    (* Table initialization: fTable_Be *)
    fTable_Be[0, 0] := 10.0000; fTable_Be[0, 1] := -9999; fTable_Be[0, 2] := 1.70333;
    fTable_Be[1, 0] := 10.1617; fTable_Be[1, 1] := -9999; fTable_Be[1, 2] := 1.71802;
    fTable_Be[2, 0] := 10.3261; fTable_Be[2, 1] := -9999; fTable_Be[2, 2] := 1.73284;
    fTable_Be[3, 0] := 10.4931; fTable_Be[3, 1] := -9999; fTable_Be[3, 2] := 1.74778;
    fTable_Be[4, 0] := 10.6628; fTable_Be[4, 1] := -9999; fTable_Be[4, 2] := 1.75737;
    fTable_Be[5, 0] := 10.8353; fTable_Be[5, 1] := -9999; fTable_Be[5, 2] := 1.76678;
    fTable_Be[6, 0] := 11.0105; fTable_Be[6, 1] := -9999; fTable_Be[6, 2] := 1.77624;
    fTable_Be[7, 0] := 11.1886; fTable_Be[7, 1] := -9999; fTable_Be[7, 2] := 1.78574;
    fTable_Be[8, 0] := 11.3696; fTable_Be[8, 1] := -9999; fTable_Be[8, 2] := 1.79530;
    fTable_Be[9, 0] := 11.5535; fTable_Be[9, 1] := -9999; fTable_Be[9, 2] := 1.80306;
    fTable_Be[10, 0] := 11.7404; fTable_Be[10, 1] := -9999; fTable_Be[10, 2] := 1.80629;
    fTable_Be[11, 0] := 11.9303; fTable_Be[11, 1] := -9999; fTable_Be[11, 2] := 1.80952;
    fTable_Be[12, 0] := 12.1232; fTable_Be[12, 1] := -9999; fTable_Be[12, 2] := 1.81276;
    fTable_Be[13, 0] := 12.3193; fTable_Be[13, 1] := -9999; fTable_Be[13, 2] := 1.81600;
    fTable_Be[14, 0] := 12.5186; fTable_Be[14, 1] := -9999; fTable_Be[14, 2] := 1.81871;
    fTable_Be[15, 0] := 12.7210; fTable_Be[15, 1] := -9999; fTable_Be[15, 2] := 1.81609;
    fTable_Be[16, 0] := 12.9268; fTable_Be[16, 1] := -9999; fTable_Be[16, 2] := 1.81347;
    fTable_Be[17, 0] := 13.1359; fTable_Be[17, 1] := -9999; fTable_Be[17, 2] := 1.80922;
    fTable_Be[18, 0] := 13.3483; fTable_Be[18, 1] := -9999; fTable_Be[18, 2] := 1.80410;
    fTable_Be[19, 0] := 13.5642; fTable_Be[19, 1] := -9999; fTable_Be[19, 2] := 1.79747;
    fTable_Be[20, 0] := 13.7836; fTable_Be[20, 1] := -9999; fTable_Be[20, 2] := 1.78729;
    fTable_Be[21, 0] := 14.0066; fTable_Be[21, 1] := -9999; fTable_Be[21, 2] := 1.77705;
    fTable_Be[22, 0] := 14.2331; fTable_Be[22, 1] := -9999; fTable_Be[22, 2] := 1.76267;
    fTable_Be[23, 0] := 14.4633; fTable_Be[23, 1] := -9999; fTable_Be[23, 2] := 1.74841;
    fTable_Be[24, 0] := 14.6972; fTable_Be[24, 1] := -9999; fTable_Be[24, 2] := 1.72956;
    fTable_Be[25, 0] := 14.9350; fTable_Be[25, 1] := -9999; fTable_Be[25, 2] := 1.71004;
    fTable_Be[26, 0] := 15.1765; fTable_Be[26, 1] := -9999; fTable_Be[26, 2] := 1.68541;
    fTable_Be[27, 0] := 15.4220; fTable_Be[27, 1] := -9999; fTable_Be[27, 2] := 1.65917;
    fTable_Be[28, 0] := 15.6714; fTable_Be[28, 1] := -9999; fTable_Be[28, 2] := 1.62778;
    fTable_Be[29, 0] := 15.9249; fTable_Be[29, 1] := -9999; fTable_Be[29, 2] := 1.59448;
    fTable_Be[30, 0] := 16.1825; fTable_Be[30, 1] := -9999; fTable_Be[30, 2] := 1.55788;
    fTable_Be[31, 0] := 16.4442; fTable_Be[31, 1] := -9999; fTable_Be[31, 2] := 1.52050;
    fTable_Be[32, 0] := 16.7102; fTable_Be[32, 1] := -9999; fTable_Be[32, 2] := 1.47675;
    fTable_Be[33, 0] := 16.9805; fTable_Be[33, 1] := -9999; fTable_Be[33, 2] := 1.43237;
    fTable_Be[34, 0] := 17.2551; fTable_Be[34, 1] := -9999; fTable_Be[34, 2] := 1.38176;
    fTable_Be[35, 0] := 17.5342; fTable_Be[35, 1] := -9999; fTable_Be[35, 2] := 1.33102;
    fTable_Be[36, 0] := 17.8178; fTable_Be[36, 1] := -9999; fTable_Be[36, 2] := 1.27265;
    fTable_Be[37, 0] := 18.1060; fTable_Be[37, 1] := -9999; fTable_Be[37, 2] := 1.22588;
    fTable_Be[38, 0] := 18.3988; fTable_Be[38, 1] := -9999; fTable_Be[38, 2] := 1.19605;
    fTable_Be[39, 0] := 18.6964; fTable_Be[39, 1] := -9999; fTable_Be[39, 2] := 1.16961;
    fTable_Be[40, 0] := 18.9988; fTable_Be[40, 1] := -9999; fTable_Be[40, 2] := 1.14509;
    fTable_Be[41, 0] := 19.3061; fTable_Be[41, 1] := 2.30967; fTable_Be[41, 2] := 1.10518;
    fTable_Be[42, 0] := 19.6184; fTable_Be[42, 1] := 2.31367; fTable_Be[42, 2] := 1.06950;
    fTable_Be[43, 0] := 19.9357; fTable_Be[43, 1] := 2.31537; fTable_Be[43, 2] := 1.03964;
    fTable_Be[44, 0] := 20.2581; fTable_Be[44, 1] := 2.31755; fTable_Be[44, 2] := 1.01722;
    fTable_Be[45, 0] := 20.5858; fTable_Be[45, 1] := 2.32374; fTable_Be[45, 2] := 0.999039;
    fTable_Be[46, 0] := 20.9187; fTable_Be[46, 1] := 2.34045; fTable_Be[46, 2] := 0.987135;
    fTable_Be[47, 0] := 21.2571; fTable_Be[47, 1] := 2.37239; fTable_Be[47, 2] := 0.952742;
    fTable_Be[48, 0] := 21.6009; fTable_Be[48, 1] := 2.38699; fTable_Be[48, 2] := 0.912693;
    fTable_Be[49, 0] := 21.9503; fTable_Be[49, 1] := 2.39600; fTable_Be[49, 2] := 0.874329;
    fTable_Be[50, 0] := 22.3053; fTable_Be[50, 1] := 2.40177; fTable_Be[50, 2] := 0.837576;
    fTable_Be[51, 0] := 22.6661; fTable_Be[51, 1] := 2.40538; fTable_Be[51, 2] := 0.802368;
    fTable_Be[52, 0] := 23.0327; fTable_Be[52, 1] := 2.40746; fTable_Be[52, 2] := 0.768641;
    fTable_Be[53, 0] := 23.4052; fTable_Be[53, 1] := 2.40846; fTable_Be[53, 2] := 0.736331;
    fTable_Be[54, 0] := 23.7838; fTable_Be[54, 1] := 2.40939; fTable_Be[54, 2] := 0.705380;
    fTable_Be[55, 0] := 24.1685; fTable_Be[55, 1] := 2.41248; fTable_Be[55, 2] := 0.675729;
    fTable_Be[56, 0] := 24.5594; fTable_Be[56, 1] := 2.41570; fTable_Be[56, 2] := 0.647325;
    fTable_Be[57, 0] := 24.9566; fTable_Be[57, 1] := 2.42027; fTable_Be[57, 2] := 0.609275;
    fTable_Be[58, 0] := 25.3602; fTable_Be[58, 1] := 2.41808; fTable_Be[58, 2] := 0.567900;
    fTable_Be[59, 0] := 25.7704; fTable_Be[59, 1] := 2.40985; fTable_Be[59, 2] := 0.529334;
    fTable_Be[60, 0] := 26.1872; fTable_Be[60, 1] := 2.39826; fTable_Be[60, 2] := 0.493388;
    fTable_Be[61, 0] := 26.6108; fTable_Be[61, 1] := 2.38435; fTable_Be[61, 2] := 0.459883;
    fTable_Be[62, 0] := 27.0412; fTable_Be[62, 1] := 2.36859; fTable_Be[62, 2] := 0.428653;
    fTable_Be[63, 0] := 27.4786; fTable_Be[63, 1] := 2.35116; fTable_Be[63, 2] := 0.399544;
    fTable_Be[64, 0] := 27.9230; fTable_Be[64, 1] := 2.33226; fTable_Be[64, 2] := 0.372411;
    fTable_Be[65, 0] := 28.3747; fTable_Be[65, 1] := 2.30996; fTable_Be[65, 2] := 0.347121;
    fTable_Be[66, 0] := 28.8336; fTable_Be[66, 1] := 2.28594; fTable_Be[66, 2] := 0.328404;
    fTable_Be[67, 0] := 29.3000; fTable_Be[67, 1] := 2.26312; fTable_Be[67, 2] := 0.315229;
    fTable_Be[68, 0] := 29.7739; fTable_Be[68, 1] := 2.24541; fTable_Be[68, 2] := 0.302582;
    fTable_Be[69, 0] := 30.2554; fTable_Be[69, 1] := 2.22901; fTable_Be[69, 2] := 0.290443;
    fTable_Be[70, 0] := 30.7448; fTable_Be[70, 1] := 2.21325; fTable_Be[70, 2] := 0.278791;
    fTable_Be[71, 0] := 31.2421; fTable_Be[71, 1] := 2.19800; fTable_Be[71, 2] := 0.267606;
    fTable_Be[72, 0] := 31.7474; fTable_Be[72, 1] := 2.18311; fTable_Be[72, 2] := 0.256870;
    fTable_Be[73, 0] := 32.2609; fTable_Be[73, 1] := 2.16844; fTable_Be[73, 2] := 0.246565;
    fTable_Be[74, 0] := 32.7827; fTable_Be[74, 1] := 2.15391; fTable_Be[74, 2] := 0.236673;
    fTable_Be[75, 0] := 33.3129; fTable_Be[75, 1] := 2.13952; fTable_Be[75, 2] := 0.227178;
    fTable_Be[76, 0] := 33.8517; fTable_Be[76, 1] := 2.12325; fTable_Be[76, 2] := 0.218064;
    fTable_Be[77, 0] := 34.3992; fTable_Be[77, 1] := 2.10677; fTable_Be[77, 2] := 0.211374;
    fTable_Be[78, 0] := 34.9556; fTable_Be[78, 1] := 2.09142; fTable_Be[78, 2] := 0.206573;
    fTable_Be[79, 0] := 35.5210; fTable_Be[79, 1] := 2.07852; fTable_Be[79, 2] := 0.201882;
    fTable_Be[80, 0] := 36.0955; fTable_Be[80, 1] := 2.06586; fTable_Be[80, 2] := 0.197297;
    fTable_Be[81, 0] := 36.6793; fTable_Be[81, 1] := 2.05353; fTable_Be[81, 2] := 0.192816;
    fTable_Be[82, 0] := 37.2726; fTable_Be[82, 1] := 2.04141; fTable_Be[82, 2] := 0.188437;
    fTable_Be[83, 0] := 37.8754; fTable_Be[83, 1] := 2.02931; fTable_Be[83, 2] := 0.184157;
    fTable_Be[84, 0] := 38.4880; fTable_Be[84, 1] := 2.01697; fTable_Be[84, 2] := 0.179975;
    fTable_Be[85, 0] := 38.9000; fTable_Be[85, 1] := 2.00799; fTable_Be[85, 2] := 0.177252;
    fTable_Be[86, 0] := 39.2000; fTable_Be[86, 1] := 2.00121; fTable_Be[86, 2] := 0.176713;
    fTable_Be[87, 0] := 39.5000; fTable_Be[87, 1] := 1.99567; fTable_Be[87, 2] := 0.176983;
    fTable_Be[88, 0] := 39.9000; fTable_Be[88, 1] := 1.98913; fTable_Be[88, 2] := 0.175827;
    fTable_Be[89, 0] := 40.0000; fTable_Be[89, 1] := 1.98733; fTable_Be[89, 2] := 0.175565;
    fTable_Be[90, 0] := 40.2760; fTable_Be[90, 1] := 1.98264; fTable_Be[90, 2] := 0.174663;
    fTable_Be[91, 0] := 40.5560; fTable_Be[91, 1] := 1.97786; fTable_Be[91, 2] := 0.174609;
    fTable_Be[92, 0] := 40.6970; fTable_Be[92, 1] := 1.97610; fTable_Be[92, 2] := 0.174013;
    fTable_Be[93, 0] := 41.1270; fTable_Be[93, 1] := 1.96960; fTable_Be[93, 2] := 0.173456;
    fTable_Be[94, 0] := 41.5660; fTable_Be[94, 1] := 1.96327; fTable_Be[94, 2] := 0.171435;
    fTable_Be[95, 0] := 42.1670; fTable_Be[95, 1] := 1.95400; fTable_Be[95, 2] := 0.170039;
    fTable_Be[96, 0] := 42.4730; fTable_Be[96, 1] := 1.94966; fTable_Be[96, 2] := 0.168799;
    fTable_Be[97, 0] := 42.9420; fTable_Be[97, 1] := 1.94280; fTable_Be[97, 2] := 0.168198;
    fTable_Be[98, 0] := 43.2600; fTable_Be[98, 1] := 1.93854; fTable_Be[98, 2] := 0.166905;
    fTable_Be[99, 0] := 43.7460; fTable_Be[99, 1] := 1.93138; fTable_Be[99, 2] := 0.165791;
    fTable_Be[100, 0] := 44.0760; fTable_Be[100, 1] := 1.92708; fTable_Be[100, 2] := 0.165390;
    fTable_Be[101, 0] := 44.4110; fTable_Be[101, 1] := 1.92291; fTable_Be[101, 2] := 0.164383;
    fTable_Be[102, 0] := 44.5810; fTable_Be[102, 1] := 1.92070; fTable_Be[102, 2] := 0.163618;
    fTable_Be[103, 0] := 44.9240; fTable_Be[103, 1] := 1.91607; fTable_Be[103, 2] := 0.162962;
    fTable_Be[104, 0] := 45.2720; fTable_Be[104, 1] := 1.91126; fTable_Be[104, 2] := 0.161326;
    fTable_Be[105, 0] := 45.4480; fTable_Be[105, 1] := 1.90903; fTable_Be[105, 2] := 0.161038;
    fTable_Be[106, 0] := 45.9850; fTable_Be[106, 1] := 1.90129; fTable_Be[106, 2] := 0.159149;
    fTable_Be[107, 0] := 46.7288; fTable_Be[107, 1] := 1.89036; fTable_Be[107, 2] := 0.157516;
    fTable_Be[108, 0] := 47.4846; fTable_Be[108, 1] := 1.87948; fTable_Be[108, 2] := 0.155990;
    fTable_Be[109, 0] := 47.6740; fTable_Be[109, 1] := 1.87667; fTable_Be[109, 2] := 0.155621;
    fTable_Be[110, 0] := 48.2650; fTable_Be[110, 1] := 1.86782; fTable_Be[110, 2] := 0.155028;
    fTable_Be[111, 0] := 48.8710; fTable_Be[111, 1] := 1.85943; fTable_Be[111, 2] := 0.155666;
    fTable_Be[112, 0] := 49.0760; fTable_Be[112, 1] := 1.85755; fTable_Be[112, 2] := 0.155951;
    fTable_Be[113, 0] := 49.2830; fTable_Be[113, 1] := 1.85503; fTable_Be[113, 2] := 0.154508;
    fTable_Be[114, 0] := 49.8930; fTable_Be[114, 1] := 1.84657; fTable_Be[114, 2] := 0.154198;
    fTable_Be[115, 0] := 50.7000; fTable_Be[115, 1] := 1.83364; fTable_Be[115, 2] := 0.155814;
    fTable_Be[116, 0] := 51.5200; fTable_Be[116, 1] := 1.82367; fTable_Be[116, 2] := 0.157447;
    fTable_Be[117, 0] := 51.9010; fTable_Be[117, 1] := 1.81956; fTable_Be[117, 2] := 0.158203;
    fTable_Be[118, 0] := 52.4010; fTable_Be[118, 1] := 1.81434; fTable_Be[118, 2] := 0.158683;
    fTable_Be[119, 0] := 53.2485; fTable_Be[119, 1] := 1.80585; fTable_Be[119, 2] := 0.158768;
    fTable_Be[120, 0] := 53.4010; fTable_Be[120, 1] := 1.80449; fTable_Be[120, 2] := 0.158784;
    fTable_Be[121, 0] := 53.9000; fTable_Be[121, 1] := 1.79914; fTable_Be[121, 2] := 0.157647;
    fTable_Be[122, 0] := 54.4010; fTable_Be[122, 1] := 1.79325; fTable_Be[122, 2] := 0.156933;
    fTable_Be[123, 0] := 54.9010; fTable_Be[123, 1] := 1.78748; fTable_Be[123, 2] := 0.157035;
    fTable_Be[124, 0] := 55.4000; fTable_Be[124, 1] := 1.78219; fTable_Be[124, 2] := 0.156125;
    fTable_Be[125, 0] := 55.9010; fTable_Be[125, 1] := 1.77644; fTable_Be[125, 2] := 0.155633;
    fTable_Be[126, 0] := 56.8052; fTable_Be[126, 1] := 1.76616; fTable_Be[126, 2] := 0.152967;
    fTable_Be[127, 0] := 56.9010; fTable_Be[127, 1] := 1.76491; fTable_Be[127, 2] := 0.152689;
    fTable_Be[128, 0] := 57.4010; fTable_Be[128, 1] := 1.75779; fTable_Be[128, 2] := 0.151560;
    fTable_Be[129, 0] := 57.9010; fTable_Be[129, 1] := 1.75138; fTable_Be[129, 2] := 0.151256;
    fTable_Be[130, 0] := 58.4000; fTable_Be[130, 1] := 1.74467; fTable_Be[130, 2] := 0.149795;
    fTable_Be[131, 0] := 59.3446; fTable_Be[131, 1] := 1.73066; fTable_Be[131, 2] := 0.148143;
    fTable_Be[132, 0] := 60.3044; fTable_Be[132, 1] := 1.71666; fTable_Be[132, 2] := 0.147555;
    fTable_Be[133, 0] := 60.9010; fTable_Be[133, 1] := 1.70803; fTable_Be[133, 2] := 0.147236;
    fTable_Be[134, 0] := 61.4010; fTable_Be[134, 1] := 1.70036; fTable_Be[134, 2] := 0.146656;
    fTable_Be[135, 0] := 62.3941; fTable_Be[135, 1] := 1.68542; fTable_Be[135, 2] := 0.147197;
    fTable_Be[136, 0] := 62.4010; fTable_Be[136, 1] := 1.68532; fTable_Be[136, 2] := 0.147201;
    fTable_Be[137, 0] := 63.4000; fTable_Be[137, 1] := 1.67044; fTable_Be[137, 2] := 0.146706;
    fTable_Be[138, 0] := 63.9020; fTable_Be[138, 1] := 1.66247; fTable_Be[138, 2] := 0.147388;
    fTable_Be[139, 0] := 64.4000; fTable_Be[139, 1] := 1.65492; fTable_Be[139, 2] := 0.147185;
    fTable_Be[140, 0] := 65.4010; fTable_Be[140, 1] := 1.63983; fTable_Be[140, 2] := 0.147806;
    fTable_Be[141, 0] := 65.9010; fTable_Be[141, 1] := 1.63182; fTable_Be[141, 2] := 0.147426;
    fTable_Be[142, 0] := 66.9669; fTable_Be[142, 1] := 1.61497; fTable_Be[142, 2] := 0.147801;
    fTable_Be[143, 0] := 68.0500; fTable_Be[143, 1] := 1.59766; fTable_Be[143, 2] := 0.147747;
    fTable_Be[144, 0] := 69.1507; fTable_Be[144, 1] := 1.57948; fTable_Be[144, 2] := 0.147404;
    fTable_Be[145, 0] := 69.4010; fTable_Be[145, 1] := 1.57524; fTable_Be[145, 2] := 0.147327;
    fTable_Be[146, 0] := 70.2340; fTable_Be[146, 1] := 1.56001; fTable_Be[146, 2] := 0.145950;
    fTable_Be[147, 0] := 71.3700; fTable_Be[147, 1] := 1.53888; fTable_Be[147, 2] := 0.145981;
    fTable_Be[148, 0] := 72.5243; fTable_Be[148, 1] := 1.51676; fTable_Be[148, 2] := 0.146011;
    fTable_Be[149, 0] := 72.5670; fTable_Be[149, 1] := 1.51586; fTable_Be[149, 2] := 0.146012;
    fTable_Be[150, 0] := 72.9000; fTable_Be[150, 1] := 1.50929; fTable_Be[150, 2] := 0.145632;
    fTable_Be[151, 0] := 73.5680; fTable_Be[151, 1] := 1.49567; fTable_Be[151, 2] := 0.146079;
    fTable_Be[152, 0] := 74.7579; fTable_Be[152, 1] := 1.47049; fTable_Be[152, 2] := 0.146106;
    fTable_Be[153, 0] := 74.9000; fTable_Be[153, 1] := 1.46741; fTable_Be[153, 2] := 0.146109;
    fTable_Be[154, 0] := 75.2350; fTable_Be[154, 1] := 1.46015; fTable_Be[154, 2] := 0.146426;
    fTable_Be[155, 0] := 75.5670; fTable_Be[155, 1] := 1.45305; fTable_Be[155, 2] := 0.146447;
    fTable_Be[156, 0] := 76.5680; fTable_Be[156, 1] := 1.43052; fTable_Be[156, 2] := 0.147310;
    fTable_Be[157, 0] := 77.2350; fTable_Be[157, 1] := 1.41539; fTable_Be[157, 2] := 0.147639;
    fTable_Be[158, 0] := 77.5670; fTable_Be[158, 1] := 1.40764; fTable_Be[158, 2] := 0.148124;
    fTable_Be[159, 0] := 77.9010; fTable_Be[159, 1] := 1.40006; fTable_Be[159, 2] := 0.148179;
    fTable_Be[160, 0] := 78.5670; fTable_Be[160, 1] := 1.38396; fTable_Be[160, 2] := 0.148938;
    fTable_Be[161, 0] := 78.9000; fTable_Be[161, 1] := 1.37631; fTable_Be[161, 2] := 0.148969;
    fTable_Be[162, 0] := 80.1761; fTable_Be[162, 1] := 1.34408; fTable_Be[162, 2] := 0.150222;
    fTable_Be[163, 0] := 80.9000; fTable_Be[163, 1] := 1.32524; fTable_Be[163, 2] := 0.150928;
    fTable_Be[164, 0] := 81.2340; fTable_Be[164, 1] := 1.31669; fTable_Be[164, 2] := 0.151099;
    fTable_Be[165, 0] := 81.5680; fTable_Be[165, 1] := 1.30817; fTable_Be[165, 2] := 0.151573;
    fTable_Be[166, 0] := 82.8873; fTable_Be[166, 1] := 1.27205; fTable_Be[166, 2] := 0.152380;
    fTable_Be[167, 0] := 83.5680; fTable_Be[167, 1] := 1.25273; fTable_Be[167, 2] := 0.152793;
    fTable_Be[168, 0] := 84.9010; fTable_Be[168, 1] := 1.21283; fTable_Be[168, 2] := 0.152919;
    fTable_Be[169, 0] := 86.2742; fTable_Be[169, 1] := 1.16875; fTable_Be[169, 2] := 0.153088;
    fTable_Be[170, 0] := 87.6696; fTable_Be[170, 1] := 1.12068; fTable_Be[170, 2] := 0.152944;
    fTable_Be[171, 0] := 89.0876; fTable_Be[171, 1] := 1.06780; fTable_Be[171, 2] := 0.152717;
    fTable_Be[172, 0] := 90.5285; fTable_Be[172, 1] := 1.00938; fTable_Be[172, 2] := 0.152457;
    fTable_Be[173, 0] := 91.9928; fTable_Be[173, 1] := 0.944630; fTable_Be[173, 2] := 0.152189;
    fTable_Be[174, 0] := 93.4807; fTable_Be[174, 1] := 0.872376; fTable_Be[174, 2] := 0.151920;
    fTable_Be[175, 0] := 94.9926; fTable_Be[175, 1] := 0.791324; fTable_Be[175, 2] := 0.151867;
    fTable_Be[176, 0] := 96.5291; fTable_Be[176, 1] := 0.699761; fTable_Be[176, 2] := 0.151828;
    fTable_Be[177, 0] := 97.5670; fTable_Be[177, 1] := 0.631310; fTable_Be[177, 2] := 0.151801;
    fTable_Be[178, 0] := 98.5680; fTable_Be[178, 1] := 0.560328; fTable_Be[178, 2] := 0.152508;
    fTable_Be[179, 0] := 98.7770; fTable_Be[179, 1] := 0.544993; fTable_Be[179, 2] := 0.152245;
    fTable_Be[180, 0] := 99.5260; fTable_Be[180, 1] := 0.486543; fTable_Be[180, 2] := 0.151861;
    fTable_Be[181, 0] := 99.9010; fTable_Be[181, 1] := 0.455599; fTable_Be[181, 2] := 0.151904;
    fTable_Be[182, 0] := 100.270; fTable_Be[182, 1] := 0.424344; fTable_Be[182, 2] := 0.151744;
    fTable_Be[183, 0] := 100.660; fTable_Be[183, 1] := 0.389731; fTable_Be[183, 2] := 0.152054;
    fTable_Be[184, 0] := 102.030; fTable_Be[184, 1] := 0.258588; fTable_Be[184, 2] := 0.151656;
    fTable_Be[185, 0] := 102.400; fTable_Be[185, 1] := 0.219148; fTable_Be[185, 2] := 0.151818;
    fTable_Be[186, 0] := 103.770; fTable_Be[186, 1] := 0.0597848; fTable_Be[186, 2] := 0.151969;
    fTable_Be[187, 0] := 104.030; fTable_Be[187, 1] := 0.0260858; fTable_Be[187, 2] := 0.152169;
    fTable_Be[188, 0] := 105.530; fTable_Be[188, 1] := -0.191568; fTable_Be[188, 2] := 0.151371;
    fTable_Be[189, 0] := 106.530; fTable_Be[189, 1] := -0.368308; fTable_Be[189, 2] := 0.151676;
    fTable_Be[190, 0] := 106.900; fTable_Be[190, 1] := -0.441904; fTable_Be[190, 2] := 0.152246;
    fTable_Be[191, 0] := 107.770; fTable_Be[191, 1] := -0.637412; fTable_Be[191, 2] := 0.154099;
    fTable_Be[192, 0] := 108.030; fTable_Be[192, 1] := -0.702374; fTable_Be[192, 2] := 0.155662;
    fTable_Be[193, 0] := 108.280; fTable_Be[193, 1] := -0.768299; fTable_Be[193, 2] := 0.156220;
    fTable_Be[194, 0] := 108.400; fTable_Be[194, 1] := -0.802126; fTable_Be[194, 2] := 0.155741;
    fTable_Be[195, 0] := 108.530; fTable_Be[195, 1] := -0.840651; fTable_Be[195, 2] := 0.156004;
    fTable_Be[196, 0] := 108.650; fTable_Be[196, 1] := -0.876311; fTable_Be[196, 2] := 0.158215;
    fTable_Be[197, 0] := 108.770; fTable_Be[197, 1] := -0.912731; fTable_Be[197, 2] := 0.158122;
    fTable_Be[198, 0] := 109.030; fTable_Be[198, 1] := -0.997553; fTable_Be[198, 2] := 0.159793;
    fTable_Be[199, 0] := 109.150; fTable_Be[199, 1] := -1.03849; fTable_Be[199, 2] := 0.161052;
    fTable_Be[200, 0] := 109.270; fTable_Be[200, 1] := -1.08113; fTable_Be[200, 2] := 0.161306;
    fTable_Be[201, 0] := 109.400; fTable_Be[201, 1] := -1.12894; fTable_Be[201, 2] := 0.163454;
    fTable_Be[202, 0] := 109.530; fTable_Be[202, 1] := -1.17915; fTable_Be[202, 2] := 0.163557;
    fTable_Be[203, 0] := 109.770; fTable_Be[203, 1] := -1.27829; fTable_Be[203, 2] := 0.165902;
    fTable_Be[204, 0] := 109.900; fTable_Be[204, 1] := -1.33524; fTable_Be[204, 2] := 0.168057;
    fTable_Be[205, 0] := 110.030; fTable_Be[205, 1] := -1.39580; fTable_Be[205, 2] := 0.168777;
    fTable_Be[206, 0] := 110.160; fTable_Be[206, 1] := -1.45968; fTable_Be[206, 2] := 0.171253;
    fTable_Be[207, 0] := 110.270; fTable_Be[207, 1] := -1.51640; fTable_Be[207, 2] := 0.172992;
    fTable_Be[208, 0] := 110.530; fTable_Be[208, 1] := -1.66366; fTable_Be[208, 2] := 0.176080;
    fTable_Be[209, 0] := 110.660; fTable_Be[209, 1] := -1.74613; fTable_Be[209, 2] := 0.179584;
    fTable_Be[210, 0] := 110.770; fTable_Be[210, 1] := -1.81926; fTable_Be[210, 2] := 0.183052;
    fTable_Be[211, 0] := 110.900; fTable_Be[211, 1] := -1.91441; fTable_Be[211, 2] := 0.183759;
    fTable_Be[212, 0] := 111.030; fTable_Be[212, 1] := -2.01892; fTable_Be[212, 2] := 0.188659;
    fTable_Be[213, 0] := 111.150; fTable_Be[213, 1] := -2.12502; fTable_Be[213, 2] := 0.191441;
    fTable_Be[214, 0] := 111.280; fTable_Be[214, 1] := -2.25725; fTable_Be[214, 2] := 0.192239;
    fTable_Be[215, 0] := 111.400; fTable_Be[215, 1] := -2.40087; fTable_Be[215, 2] := 0.199075;
    fTable_Be[216, 0] := 111.530; fTable_Be[216, 1] := -2.58708; fTable_Be[216, 2] := 0.209517;
    fTable_Be[217, 0] := 111.600; fTable_Be[217, 1] := -2.70637; fTable_Be[217, 2] := 0.223326;
    fTable_Be[218, 0] := 111.800; fTable_Be[218, 1] := -3.21583; fTable_Be[218, 2] := 0.378238;
    fTable_Be[219, 0] := 112.000; fTable_Be[219, 1] := -3.42252; fTable_Be[219, 2] := 1.03860;
    fTable_Be[220, 0] := 112.250; fTable_Be[220, 1] := -3.41684; fTable_Be[220, 2] := 1.38190;
    fTable_Be[221, 0] := 112.500; fTable_Be[221, 1] := -3.59292; fTable_Be[221, 2] := 1.57501;
    fTable_Be[222, 0] := 112.750; fTable_Be[222, 1] := -3.95038; fTable_Be[222, 2] := 2.03965;
    fTable_Be[223, 0] := 113.000; fTable_Be[223, 1] := -3.99197; fTable_Be[223, 2] := 3.05986;
    fTable_Be[224, 0] := 113.250; fTable_Be[224, 1] := -3.32582; fTable_Be[224, 2] := 4.01793;
    fTable_Be[225, 0] := 113.500; fTable_Be[225, 1] := -2.38510; fTable_Be[225, 2] := 4.15418;
    fTable_Be[226, 0] := 113.750; fTable_Be[226, 1] := -1.77257; fTable_Be[226, 2] := 3.84564;
    fTable_Be[227, 0] := 114.000; fTable_Be[227, 1] := -1.49267; fTable_Be[227, 2] := 3.56793;
    fTable_Be[228, 0] := 114.250; fTable_Be[228, 1] := -1.40646; fTable_Be[228, 2] := 3.26353;
    fTable_Be[229, 0] := 114.500; fTable_Be[229, 1] := -1.45558; fTable_Be[229, 2] := 3.11127;
    fTable_Be[230, 0] := 114.750; fTable_Be[230, 1] := -1.51462; fTable_Be[230, 2] := 3.06546;
    fTable_Be[231, 0] := 115.000; fTable_Be[231, 1] := -1.58085; fTable_Be[231, 2] := 3.03372;
    fTable_Be[232, 0] := 115.500; fTable_Be[232, 1] := -1.68141; fTable_Be[232, 2] := 3.14487;
    fTable_Be[233, 0] := 115.750; fTable_Be[233, 1] := -1.68766; fTable_Be[233, 2] := 3.23324;
    fTable_Be[234, 0] := 116.000; fTable_Be[234, 1] := -1.67443; fTable_Be[234, 2] := 3.28469;
    fTable_Be[235, 0] := 116.250; fTable_Be[235, 1] := -1.69668; fTable_Be[235, 2] := 3.30771;
    fTable_Be[236, 0] := 116.500; fTable_Be[236, 1] := -1.74476; fTable_Be[236, 2] := 3.36223;
    fTable_Be[237, 0] := 116.750; fTable_Be[237, 1] := -1.84100; fTable_Be[237, 2] := 3.42546;
    fTable_Be[238, 0] := 117.000; fTable_Be[238, 1] := -1.91971; fTable_Be[238, 2] := 3.58866;
    fTable_Be[239, 0] := 117.250; fTable_Be[239, 1] := -2.01798; fTable_Be[239, 2] := 3.75177;
    fTable_Be[240, 0] := 117.500; fTable_Be[240, 1] := -2.09181; fTable_Be[240, 2] := 4.02099;
    fTable_Be[241, 0] := 117.750; fTable_Be[241, 1] := -1.98599; fTable_Be[241, 2] := 4.48576;
    fTable_Be[242, 0] := 118.000; fTable_Be[242, 1] := -1.69069; fTable_Be[242, 2] := 4.69519;
    fTable_Be[243, 0] := 118.250; fTable_Be[243, 1] := -1.41511; fTable_Be[243, 2] := 4.80543;
    fTable_Be[244, 0] := 118.500; fTable_Be[244, 1] := -1.17170; fTable_Be[244, 2] := 4.79021;
    fTable_Be[245, 0] := 118.750; fTable_Be[245, 1] := -1.03307; fTable_Be[245, 2] := 4.76242;
    fTable_Be[246, 0] := 119.000; fTable_Be[246, 1] := -0.919695; fTable_Be[246, 2] := 4.72326;
    fTable_Be[247, 0] := 119.250; fTable_Be[247, 1] := -0.899806; fTable_Be[247, 2] := 4.70943;
    fTable_Be[248, 0] := 119.500; fTable_Be[248, 1] := -0.833607; fTable_Be[248, 2] := 4.73952;
    fTable_Be[249, 0] := 120.500; fTable_Be[249, 1] := -0.607801; fTable_Be[249, 2] := 5.01171;
    fTable_Be[250, 0] := 121.000; fTable_Be[250, 1] := -0.546931; fTable_Be[250, 2] := 4.97342;
    fTable_Be[251, 0] := 121.500; fTable_Be[251, 1] := -0.418154; fTable_Be[251, 2] := 5.37885;
    fTable_Be[252, 0] := 122.000; fTable_Be[252, 1] := -0.0951663; fTable_Be[252, 2] := 5.50733;
    fTable_Be[253, 0] := 122.500; fTable_Be[253, 1] := 0.195563; fTable_Be[253, 2] := 5.47638;
    fTable_Be[254, 0] := 123.000; fTable_Be[254, 1] := 0.287270; fTable_Be[254, 2] := 5.41101;
    fTable_Be[255, 0] := 123.500; fTable_Be[255, 1] := 0.285511; fTable_Be[255, 2] := 5.46448;
    fTable_Be[256, 0] := 124.000; fTable_Be[256, 1] := 0.326778; fTable_Be[256, 2] := 5.80078;
    fTable_Be[257, 0] := 125.000; fTable_Be[257, 1] := 0.899833; fTable_Be[257, 2] := 6.30269;
    fTable_Be[258, 0] := 125.500; fTable_Be[258, 1] := 1.34102; fTable_Be[258, 2] := 6.64803;
    fTable_Be[259, 0] := 126.000; fTable_Be[259, 1] := 1.95659; fTable_Be[259, 2] := 6.68559;
    fTable_Be[260, 0] := 126.500; fTable_Be[260, 1] := 2.54905; fTable_Be[260, 2] := 6.64790;
    fTable_Be[261, 0] := 127.000; fTable_Be[261, 1] := 3.16414; fTable_Be[261, 2] := 6.40082;
    fTable_Be[262, 0] := 127.500; fTable_Be[262, 1] := 3.67151; fTable_Be[262, 2] := 6.01367;
    fTable_Be[263, 0] := 128.000; fTable_Be[263, 1] := 3.96394; fTable_Be[263, 2] := 5.39328;
    fTable_Be[264, 0] := 128.500; fTable_Be[264, 1] := 4.07172; fTable_Be[264, 2] := 5.00813;
    fTable_Be[265, 0] := 129.000; fTable_Be[265, 1] := 4.14772; fTable_Be[265, 2] := 4.55903;
    fTable_Be[266, 0] := 129.500; fTable_Be[266, 1] := 4.13409; fTable_Be[266, 2] := 4.20865;
    fTable_Be[267, 0] := 130.000; fTable_Be[267, 1] := 4.07072; fTable_Be[267, 2] := 3.82730;
    fTable_Be[268, 0] := 130.500; fTable_Be[268, 1] := 3.96867; fTable_Be[268, 2] := 3.59578;
    fTable_Be[269, 0] := 131.000; fTable_Be[269, 1] := 3.81583; fTable_Be[269, 2] := 3.26529;
    fTable_Be[270, 0] := 131.500; fTable_Be[270, 1] := 3.62226; fTable_Be[270, 2] := 3.15721;
    fTable_Be[271, 0] := 132.000; fTable_Be[271, 1] := 3.45638; fTable_Be[271, 2] := 3.02786;
    fTable_Be[272, 0] := 133.000; fTable_Be[272, 1] := 3.17671; fTable_Be[272, 2] := 2.92660;
    fTable_Be[273, 0] := 133.500; fTable_Be[273, 1] := 3.07605; fTable_Be[273, 2] := 2.93560;
    fTable_Be[274, 0] := 134.000; fTable_Be[274, 1] := 3.00843; fTable_Be[274, 2] := 2.93684;
    fTable_Be[275, 0] := 134.500; fTable_Be[275, 1] := 2.96221; fTable_Be[275, 2] := 2.94578;
    fTable_Be[276, 0] := 135.500; fTable_Be[276, 1] := 2.89396; fTable_Be[276, 2] := 2.93779;
    fTable_Be[277, 0] := 136.000; fTable_Be[277, 1] := 2.87584; fTable_Be[277, 2] := 2.94397;
    fTable_Be[278, 0] := 136.500; fTable_Be[278, 1] := 2.86874; fTable_Be[278, 2] := 2.93959;
    fTable_Be[279, 0] := 137.500; fTable_Be[279, 1] := 2.85627; fTable_Be[279, 2] := 2.89893;
    fTable_Be[280, 0] := 138.000; fTable_Be[280, 1] := 2.83336; fTable_Be[280, 2] := 2.87398;
    fTable_Be[281, 0] := 138.500; fTable_Be[281, 1] := 2.81506; fTable_Be[281, 2] := 2.87098;
    fTable_Be[282, 0] := 139.000; fTable_Be[282, 1] := 2.79734; fTable_Be[282, 2] := 2.84887;
    fTable_Be[283, 0] := 140.000; fTable_Be[283, 1] := 2.73715; fTable_Be[283, 2] := 2.83539;
    fTable_Be[284, 0] := 141.000; fTable_Be[284, 1] := 2.69982; fTable_Be[284, 2] := 2.87711;
    fTable_Be[285, 0] := 141.500; fTable_Be[285, 1] := 2.70638; fTable_Be[285, 2] := 2.90329;
    fTable_Be[286, 0] := 142.000; fTable_Be[286, 1] := 2.71550; fTable_Be[286, 2] := 2.90287;
    fTable_Be[287, 0] := 142.500; fTable_Be[287, 1] := 2.72019; fTable_Be[287, 2] := 2.91465;
    fTable_Be[288, 0] := 143.000; fTable_Be[288, 1] := 2.72987; fTable_Be[288, 2] := 2.91685;
    fTable_Be[289, 0] := 143.500; fTable_Be[289, 1] := 2.74333; fTable_Be[289, 2] := 2.92650;
    fTable_Be[290, 0] := 144.000; fTable_Be[290, 1] := 2.75592; fTable_Be[290, 2] := 2.91495;
    fTable_Be[291, 0] := 144.500; fTable_Be[291, 1] := 2.76383; fTable_Be[291, 2] := 2.91585;
    fTable_Be[292, 0] := 145.000; fTable_Be[292, 1] := 2.76841; fTable_Be[292, 2] := 2.90262;
    fTable_Be[293, 0] := 145.500; fTable_Be[293, 1] := 2.77007; fTable_Be[293, 2] := 2.90346;
    fTable_Be[294, 0] := 146.000; fTable_Be[294, 1] := 2.76964; fTable_Be[294, 2] := 2.89577;
    fTable_Be[295, 0] := 146.500; fTable_Be[295, 1] := 2.76561; fTable_Be[295, 2] := 2.89537;
    fTable_Be[296, 0] := 148.000; fTable_Be[296, 1] := 2.76343; fTable_Be[296, 2] := 2.93154;
    fTable_Be[297, 0] := 148.500; fTable_Be[297, 1] := 2.77483; fTable_Be[297, 2] := 2.94822;
    fTable_Be[298, 0] := 149.000; fTable_Be[298, 1] := 2.78740; fTable_Be[298, 2] := 2.95243;
    fTable_Be[299, 0] := 150.000; fTable_Be[299, 1] := 2.81919; fTable_Be[299, 2] := 2.98597;
    fTable_Be[300, 0] := 151.000; fTable_Be[300, 1] := 2.85322; fTable_Be[300, 2] := 2.98029;
    fTable_Be[301, 0] := 152.000; fTable_Be[301, 1] := 2.86818; fTable_Be[301, 2] := 2.98203;
    fTable_Be[302, 0] := 153.000; fTable_Be[302, 1] := 2.89266; fTable_Be[302, 2] := 3.01367;
    fTable_Be[303, 0] := 153.500; fTable_Be[303, 1] := 2.89847; fTable_Be[303, 2] := 3.01671;
    fTable_Be[304, 0] := 155.000; fTable_Be[304, 1] := 2.93623; fTable_Be[304, 2] := 3.06074;
    fTable_Be[305, 0] := 155.500; fTable_Be[305, 1] := 2.96092; fTable_Be[305, 2] := 3.08803;
    fTable_Be[306, 0] := 156.500; fTable_Be[306, 1] := 3.01251; fTable_Be[306, 2] := 3.12840;
    fTable_Be[307, 0] := 157.000; fTable_Be[307, 1] := 3.04430; fTable_Be[307, 2] := 3.14926;
    fTable_Be[308, 0] := 157.500; fTable_Be[308, 1] := 3.08675; fTable_Be[308, 2] := 3.17679;
    fTable_Be[309, 0] := 158.000; fTable_Be[309, 1] := 3.13492; fTable_Be[309, 2] := 3.18715;
    fTable_Be[310, 0] := 159.000; fTable_Be[310, 1] := 3.22830; fTable_Be[310, 2] := 3.19053;
    fTable_Be[311, 0] := 160.000; fTable_Be[311, 1] := 3.32359; fTable_Be[311, 2] := 3.19716;
    fTable_Be[312, 0] := 160.500; fTable_Be[312, 1] := 3.37652; fTable_Be[312, 2] := 3.19224;
    fTable_Be[313, 0] := 161.500; fTable_Be[313, 1] := 3.48313; fTable_Be[313, 2] := 3.16079;
    fTable_Be[314, 0] := 162.000; fTable_Be[314, 1] := 3.53440; fTable_Be[314, 2] := 3.15119;
    fTable_Be[315, 0] := 163.000; fTable_Be[315, 1] := 3.64004; fTable_Be[315, 2] := 3.07868;
    fTable_Be[316, 0] := 164.500; fTable_Be[316, 1] := 3.74596; fTable_Be[316, 2] := 2.93822;
    fTable_Be[317, 0] := 165.500; fTable_Be[317, 1] := 3.78278; fTable_Be[317, 2] := 2.85215;
    fTable_Be[318, 0] := 166.000; fTable_Be[318, 1] := 3.79484; fTable_Be[318, 2] := 2.81725;
    fTable_Be[319, 0] := 167.000; fTable_Be[319, 1] := 3.82135; fTable_Be[319, 2] := 2.73264;
    fTable_Be[320, 0] := 167.500; fTable_Be[320, 1] := 3.82362; fTable_Be[320, 2] := 2.69680;
    fTable_Be[321, 0] := 168.000; fTable_Be[321, 1] := 3.81959; fTable_Be[321, 2] := 2.65488;
    fTable_Be[322, 0] := 169.500; fTable_Be[322, 1] := 3.80124; fTable_Be[322, 2] := 2.57094;
    fTable_Be[323, 0] := 170.000; fTable_Be[323, 1] := 3.79268; fTable_Be[323, 2] := 2.55180;
    fTable_Be[324, 0] := 170.500; fTable_Be[324, 1] := 3.78838; fTable_Be[324, 2] := 2.54214;
    fTable_Be[325, 0] := 171.000; fTable_Be[325, 1] := 3.78748; fTable_Be[325, 2] := 2.52605;
    fTable_Be[326, 0] := 171.500; fTable_Be[326, 1] := 3.78804; fTable_Be[326, 2] := 2.51896;
    fTable_Be[327, 0] := 172.990; fTable_Be[327, 1] := 3.80814; fTable_Be[327, 2] := 2.47360;
    fTable_Be[328, 0] := 173.990; fTable_Be[328, 1] := 3.80347; fTable_Be[328, 2] := 2.43390;
    fTable_Be[329, 0] := 174.500; fTable_Be[329, 1] := 3.81339; fTable_Be[329, 2] := 2.43394;
    fTable_Be[330, 0] := 175.510; fTable_Be[330, 1] := 3.82900; fTable_Be[330, 2] := 2.40213;
    fTable_Be[331, 0] := 176.000; fTable_Be[331, 1] := 3.83339; fTable_Be[331, 2] := 2.38083;
    fTable_Be[332, 0] := 176.500; fTable_Be[332, 1] := 3.83871; fTable_Be[332, 2] := 2.36562;
    fTable_Be[333, 0] := 177.510; fTable_Be[333, 1] := 3.85216; fTable_Be[333, 2] := 2.32073;
    fTable_Be[334, 0] := 178.000; fTable_Be[334, 1] := 3.84430; fTable_Be[334, 2] := 2.28306;
    fTable_Be[335, 0] := 178.500; fTable_Be[335, 1] := 3.84361; fTable_Be[335, 2] := 2.27434;
    fTable_Be[336, 0] := 180.000; fTable_Be[336, 1] := 3.79942; fTable_Be[336, 2] := 2.22984;
    fTable_Be[337, 0] := 181.000; fTable_Be[337, 1] := 3.78489; fTable_Be[337, 2] := 2.22505;
    fTable_Be[338, 0] := 181.510; fTable_Be[338, 1] := 3.78464; fTable_Be[338, 2] := 2.22872;
    fTable_Be[339, 0] := 182.000; fTable_Be[339, 1] := 3.77923; fTable_Be[339, 2] := 2.21064;
    fTable_Be[340, 0] := 183.500; fTable_Be[340, 1] := 3.77455; fTable_Be[340, 2] := 2.19974;
    fTable_Be[341, 0] := 184.490; fTable_Be[341, 1] := 3.77588; fTable_Be[341, 2] := 2.18992;
    fTable_Be[342, 0] := 187.474; fTable_Be[342, 1] := 3.78737; fTable_Be[342, 2] := 2.16785;
    fTable_Be[343, 0] := 187.500; fTable_Be[343, 1] := 3.78737; fTable_Be[343, 2] := 2.16766;
    fTable_Be[344, 0] := 188.000; fTable_Be[344, 1] := 3.77910; fTable_Be[344, 2] := 2.15580;
    fTable_Be[345, 0] := 188.500; fTable_Be[345, 1] := 3.77675; fTable_Be[345, 2] := 2.16037;
    fTable_Be[346, 0] := 189.000; fTable_Be[346, 1] := 3.77711; fTable_Be[346, 2] := 2.15869;
    fTable_Be[347, 0] := 190.000; fTable_Be[347, 1] := 3.78555; fTable_Be[347, 2] := 2.16413;
    fTable_Be[348, 0] := 190.500; fTable_Be[348, 1] := 3.79166; fTable_Be[348, 2] := 2.15995;
    fTable_Be[349, 0] := 191.000; fTable_Be[349, 1] := 3.79603; fTable_Be[349, 2] := 2.16059;
    fTable_Be[350, 0] := 192.000; fTable_Be[350, 1] := 3.80715; fTable_Be[350, 2] := 2.14936;
    fTable_Be[351, 0] := 193.510; fTable_Be[351, 1] := 3.82898; fTable_Be[351, 2] := 2.14231;
    fTable_Be[352, 0] := 194.000; fTable_Be[352, 1] := 3.83942; fTable_Be[352, 2] := 2.13531;
    fTable_Be[353, 0] := 194.500; fTable_Be[353, 1] := 3.84007; fTable_Be[353, 2] := 2.11653;
    fTable_Be[354, 0] := 195.000; fTable_Be[354, 1] := 3.83469; fTable_Be[354, 2] := 2.11378;
    fTable_Be[355, 0] := 195.500; fTable_Be[355, 1] := 3.83653; fTable_Be[355, 2] := 2.11602;
    fTable_Be[356, 0] := 196.500; fTable_Be[356, 1] := 3.84812; fTable_Be[356, 2] := 2.10677;
    fTable_Be[357, 0] := 197.500; fTable_Be[357, 1] := 3.85281; fTable_Be[357, 2] := 2.09245;
    fTable_Be[358, 0] := 199.010; fTable_Be[358, 1] := 3.86036; fTable_Be[358, 2] := 2.09404;
    fTable_Be[359, 0] := 200.000; fTable_Be[359, 1] := 3.87172; fTable_Be[359, 2] := 2.08193;
    fTable_Be[360, 0] := 201.500; fTable_Be[360, 1] := 3.88191; fTable_Be[360, 2] := 2.07385;
    fTable_Be[361, 0] := 203.000; fTable_Be[361, 1] := 3.89450; fTable_Be[361, 2] := 2.07146;
    fTable_Be[362, 0] := 204.500; fTable_Be[362, 1] := 3.92105; fTable_Be[362, 2] := 2.06855;
    fTable_Be[363, 0] := 207.000; fTable_Be[363, 1] := 3.96780; fTable_Be[363, 2] := 2.04405;
    fTable_Be[364, 0] := 207.500; fTable_Be[364, 1] := 3.97172; fTable_Be[364, 2] := 2.03179;
    fTable_Be[365, 0] := 208.010; fTable_Be[365, 1] := 3.97628; fTable_Be[365, 2] := 2.03019;
    fTable_Be[366, 0] := 208.500; fTable_Be[366, 1] := 3.97935; fTable_Be[366, 2] := 2.02063;
    fTable_Be[367, 0] := 210.500; fTable_Be[367, 1] := 4.00635; fTable_Be[367, 2] := 2.00156;
    fTable_Be[368, 0] := 212.000; fTable_Be[368, 1] := 4.02425; fTable_Be[368, 2] := 1.97791;
    fTable_Be[369, 0] := 212.500; fTable_Be[369, 1] := 4.02760; fTable_Be[369, 2] := 1.97716;
    fTable_Be[370, 0] := 213.000; fTable_Be[370, 1] := 4.03863; fTable_Be[370, 2] := 1.96995;
    fTable_Be[371, 0] := 213.500; fTable_Be[371, 1] := 4.04264; fTable_Be[371, 2] := 1.95601;
    fTable_Be[372, 0] := 214.500; fTable_Be[372, 1] := 4.04244; fTable_Be[372, 2] := 1.94417;
    fTable_Be[373, 0] := 215.000; fTable_Be[373, 1] := 4.04818; fTable_Be[373, 2] := 1.94719;
    fTable_Be[374, 0] := 215.500; fTable_Be[374, 1] := 4.05146; fTable_Be[374, 2] := 1.93625;
    fTable_Be[375, 0] := 217.000; fTable_Be[375, 1] := 4.07177; fTable_Be[375, 2] := 1.91827;
    fTable_Be[376, 0] := 218.000; fTable_Be[376, 1] := 4.07937; fTable_Be[376, 2] := 1.90175;
    fTable_Be[377, 0] := 219.000; fTable_Be[377, 1] := 4.08572; fTable_Be[377, 2] := 1.89162;
    fTable_Be[378, 0] := 220.000; fTable_Be[378, 1] := 4.09161; fTable_Be[378, 2] := 1.87778;
    fTable_Be[379, 0] := 220.500; fTable_Be[379, 1] := 4.09066; fTable_Be[379, 2] := 1.87308;
    fTable_Be[380, 0] := 221.000; fTable_Be[380, 1] := 4.09659; fTable_Be[380, 2] := 1.87799;
    fTable_Be[381, 0] := 221.500; fTable_Be[381, 1] := 4.10445; fTable_Be[381, 2] := 1.86891;
    fTable_Be[382, 0] := 222.000; fTable_Be[382, 1] := 4.11052; fTable_Be[382, 2] := 1.86480;
    fTable_Be[383, 0] := 222.500; fTable_Be[383, 1] := 4.11500; fTable_Be[383, 2] := 1.85638;
    fTable_Be[384, 0] := 223.000; fTable_Be[384, 1] := 4.12075; fTable_Be[384, 2] := 1.85152;
    fTable_Be[385, 0] := 223.500; fTable_Be[385, 1] := 4.12176; fTable_Be[385, 2] := 1.84131;
    fTable_Be[386, 0] := 224.000; fTable_Be[386, 1] := 4.12134; fTable_Be[386, 2] := 1.83756;
    fTable_Be[387, 0] := 224.500; fTable_Be[387, 1] := 4.12348; fTable_Be[387, 2] := 1.84253;
    fTable_Be[388, 0] := 226.000; fTable_Be[388, 1] := 4.15704; fTable_Be[388, 2] := 1.82599;
    fTable_Be[389, 0] := 226.490; fTable_Be[389, 1] := 4.16101; fTable_Be[389, 2] := 1.81782;
    fTable_Be[390, 0] := 227.500; fTable_Be[390, 1] := 4.17850; fTable_Be[390, 2] := 1.80946;
    fTable_Be[391, 0] := 228.000; fTable_Be[391, 1] := 4.19190; fTable_Be[391, 2] := 1.79537;
    fTable_Be[392, 0] := 228.500; fTable_Be[392, 1] := 4.19439; fTable_Be[392, 2] := 1.77053;
    fTable_Be[393, 0] := 229.000; fTable_Be[393, 1] := 4.19072; fTable_Be[393, 2] := 1.76739;
    fTable_Be[394, 0] := 229.500; fTable_Be[394, 1] := 4.19374; fTable_Be[394, 2] := 1.75778;
    fTable_Be[395, 0] := 230.500; fTable_Be[395, 1] := 4.19691; fTable_Be[395, 2] := 1.74263;
    fTable_Be[396, 0] := 231.000; fTable_Be[396, 1] := 4.20734; fTable_Be[396, 2] := 1.73860;
    fTable_Be[397, 0] := 231.500; fTable_Be[397, 1] := 4.21071; fTable_Be[397, 2] := 1.72476;
    fTable_Be[398, 0] := 232.000; fTable_Be[398, 1] := 4.21210; fTable_Be[398, 2] := 1.70717;
    fTable_Be[399, 0] := 234.500; fTable_Be[399, 1] := 4.21500; fTable_Be[399, 2] := 1.66650;
    fTable_Be[400, 0] := 235.000; fTable_Be[400, 1] := 4.20480; fTable_Be[400, 2] := 1.65173;
    fTable_Be[401, 0] := 235.500; fTable_Be[401, 1] := 4.20096; fTable_Be[401, 2] := 1.64949;
    fTable_Be[402, 0] := 236.500; fTable_Be[402, 1] := 4.20132; fTable_Be[402, 2] := 1.65027;
    fTable_Be[403, 0] := 237.500; fTable_Be[403, 1] := 4.20371; fTable_Be[403, 2] := 1.63115;
    fTable_Be[404, 0] := 238.000; fTable_Be[404, 1] := 4.20288; fTable_Be[404, 2] := 1.62857;
    fTable_Be[405, 0] := 238.500; fTable_Be[405, 1] := 4.20322; fTable_Be[405, 2] := 1.62029;
    fTable_Be[406, 0] := 239.500; fTable_Be[406, 1] := 4.20097; fTable_Be[406, 2] := 1.61693;
    fTable_Be[407, 0] := 240.000; fTable_Be[407, 1] := 4.20624; fTable_Be[407, 2] := 1.61172;
    fTable_Be[408, 0] := 240.500; fTable_Be[408, 1] := 4.20812; fTable_Be[408, 2] := 1.60246;
    fTable_Be[409, 0] := 241.000; fTable_Be[409, 1] := 4.21110; fTable_Be[409, 2] := 1.59846;
    fTable_Be[410, 0] := 241.500; fTable_Be[410, 1] := 4.20782; fTable_Be[410, 2] := 1.58125;
    fTable_Be[411, 0] := 242.000; fTable_Be[411, 1] := 4.19755; fTable_Be[411, 2] := 1.57866;
    fTable_Be[412, 0] := 242.500; fTable_Be[412, 1] := 4.19930; fTable_Be[412, 2] := 1.58572;
    fTable_Be[413, 0] := 243.500; fTable_Be[413, 1] := 4.21118; fTable_Be[413, 2] := 1.57948;
    fTable_Be[414, 0] := 244.000; fTable_Be[414, 1] := 4.20763; fTable_Be[414, 2] := 1.56140;
    fTable_Be[415, 0] := 244.500; fTable_Be[415, 1] := 4.20246; fTable_Be[415, 2] := 1.56099;
    fTable_Be[416, 0] := 245.000; fTable_Be[416, 1] := 4.19678; fTable_Be[416, 2] := 1.55568;
    fTable_Be[417, 0] := 246.000; fTable_Be[417, 1] := 4.19512; fTable_Be[417, 2] := 1.55713;
    fTable_Be[418, 0] := 246.500; fTable_Be[418, 1] := 4.19511; fTable_Be[418, 2] := 1.55644;
    fTable_Be[419, 0] := 247.500; fTable_Be[419, 1] := 4.19613; fTable_Be[419, 2] := 1.55114;
    fTable_Be[420, 0] := 248.500; fTable_Be[420, 1] := 4.18859; fTable_Be[420, 2] := 1.55086;
    fTable_Be[421, 0] := 248.990; fTable_Be[421, 1] := 4.19626; fTable_Be[421, 2] := 1.56821;
    fTable_Be[422, 0] := 249.500; fTable_Be[422, 1] := 4.21213; fTable_Be[422, 2] := 1.56785;
    fTable_Be[423, 0] := 250.000; fTable_Be[423, 1] := 4.22653; fTable_Be[423, 2] := 1.55043;
    fTable_Be[424, 0] := 251.540; fTable_Be[424, 1] := 4.26661; fTable_Be[424, 2] := 1.54085;
    fTable_Be[425, 0] := 255.608; fTable_Be[425, 1] := 4.25156; fTable_Be[425, 2] := 1.50042;
    fTable_Be[426, 0] := 259.743; fTable_Be[426, 1] := 4.26764; fTable_Be[426, 2] := 1.46106;
    fTable_Be[427, 0] := 263.944; fTable_Be[427, 1] := 4.28045; fTable_Be[427, 2] := 1.42272;
    fTable_Be[428, 0] := 268.213; fTable_Be[428, 1] := 4.29117; fTable_Be[428, 2] := 1.38539;
    fTable_Be[429, 0] := 272.551; fTable_Be[429, 1] := 4.30032; fTable_Be[429, 2] := 1.34904;
    fTable_Be[430, 0] := 276.959; fTable_Be[430, 1] := 4.30821; fTable_Be[430, 2] := 1.31364;
    fTable_Be[431, 0] := 281.439; fTable_Be[431, 1] := 4.31501; fTable_Be[431, 2] := 1.27917;
    fTable_Be[432, 0] := 285.991; fTable_Be[432, 1] := 4.32087; fTable_Be[432, 2] := 1.24561;
    fTable_Be[433, 0] := 290.617; fTable_Be[433, 1] := 4.32588; fTable_Be[433, 2] := 1.21293;
    fTable_Be[434, 0] := 295.317; fTable_Be[434, 1] := 4.33013; fTable_Be[434, 2] := 1.18110;
    fTable_Be[435, 0] := 300.094; fTable_Be[435, 1] := 4.33368; fTable_Be[435, 2] := 1.15011;
    fTable_Be[436, 0] := 304.947; fTable_Be[436, 1] := 4.33653; fTable_Be[436, 2] := 1.11993;
    fTable_Be[437, 0] := 309.880; fTable_Be[437, 1] := 4.33874; fTable_Be[437, 2] := 1.09055;
    fTable_Be[438, 0] := 314.892; fTable_Be[438, 1] := 4.34029; fTable_Be[438, 2] := 1.06193;
    fTable_Be[439, 0] := 319.985; fTable_Be[439, 1] := 4.34126; fTable_Be[439, 2] := 1.03488;
    fTable_Be[440, 0] := 325.160; fTable_Be[440, 1] := 4.34227; fTable_Be[440, 2] := 1.00851;
    fTable_Be[441, 0] := 330.420; fTable_Be[441, 1] := 4.34307; fTable_Be[441, 2] := 0.982821;
    fTable_Be[442, 0] := 335.764; fTable_Be[442, 1] := 4.34364; fTable_Be[442, 2] := 0.957781;
    fTable_Be[443, 0] := 341.195; fTable_Be[443, 1] := 4.34399; fTable_Be[443, 2] := 0.933380;
    fTable_Be[444, 0] := 346.713; fTable_Be[444, 1] := 4.34413; fTable_Be[444, 2] := 0.909600;
    fTable_Be[445, 0] := 352.321; fTable_Be[445, 1] := 4.34408; fTable_Be[445, 2] := 0.886427;
    fTable_Be[446, 0] := 358.020; fTable_Be[446, 1] := 4.34387; fTable_Be[446, 2] := 0.863843;
    fTable_Be[447, 0] := 363.810; fTable_Be[447, 1] := 4.34352; fTable_Be[447, 2] := 0.841835;
    fTable_Be[448, 0] := 369.695; fTable_Be[448, 1] := 4.34307; fTable_Be[448, 2] := 0.820388;
    fTable_Be[449, 0] := 375.674; fTable_Be[449, 1] := 4.34247; fTable_Be[449, 2] := 0.799486;
    fTable_Be[450, 0] := 381.750; fTable_Be[450, 1] := 4.34234; fTable_Be[450, 2] := 0.779118;
    fTable_Be[451, 0] := 387.925; fTable_Be[451, 1] := 4.34238; fTable_Be[451, 2] := 0.759267;
    fTable_Be[452, 0] := 394.199; fTable_Be[452, 1] := 4.34228; fTable_Be[452, 2] := 0.738576;
    fTable_Be[453, 0] := 400.575; fTable_Be[453, 1] := 4.34177; fTable_Be[453, 2] := 0.718448;
    fTable_Be[454, 0] := 407.054; fTable_Be[454, 1] := 4.34059; fTable_Be[454, 2] := 0.697922;
    fTable_Be[455, 0] := 413.638; fTable_Be[455, 1] := 4.33897; fTable_Be[455, 2] := 0.677984;
    fTable_Be[456, 0] := 420.328; fTable_Be[456, 1] := 4.33688; fTable_Be[456, 2] := 0.658616;
    fTable_Be[457, 0] := 427.126; fTable_Be[457, 1] := 4.33438; fTable_Be[457, 2] := 0.639799;
    fTable_Be[458, 0] := 434.035; fTable_Be[458, 1] := 4.33165; fTable_Be[458, 2] := 0.621521;
    fTable_Be[459, 0] := 441.055; fTable_Be[459, 1] := 4.32870; fTable_Be[459, 2] := 0.603766;
    fTable_Be[460, 0] := 448.189; fTable_Be[460, 1] := 4.32557; fTable_Be[460, 2] := 0.586516;
    fTable_Be[461, 0] := 455.438; fTable_Be[461, 1] := 4.32228; fTable_Be[461, 2] := 0.569761;
    fTable_Be[462, 0] := 462.804; fTable_Be[462, 1] := 4.31886; fTable_Be[462, 2] := 0.553484;
    fTable_Be[463, 0] := 470.290; fTable_Be[463, 1] := 4.31532; fTable_Be[463, 2] := 0.537671;
    fTable_Be[464, 0] := 477.896; fTable_Be[464, 1] := 4.31169; fTable_Be[464, 2] := 0.522311;
    fTable_Be[465, 0] := 485.626; fTable_Be[465, 1] := 4.30798; fTable_Be[465, 2] := 0.507390;
    fTable_Be[466, 0] := 493.480; fTable_Be[466, 1] := 4.30421; fTable_Be[466, 2] := 0.492894;
    fTable_Be[467, 0] := 501.462; fTable_Be[467, 1] := 4.30038; fTable_Be[467, 2] := 0.478813;
    fTable_Be[468, 0] := 509.573; fTable_Be[468, 1] := 4.29651; fTable_Be[468, 2] := 0.465133;
    fTable_Be[469, 0] := 517.815; fTable_Be[469, 1] := 4.29262; fTable_Be[469, 2] := 0.451845;
    fTable_Be[470, 0] := 526.190; fTable_Be[470, 1] := 4.28871; fTable_Be[470, 2] := 0.438937;
    fTable_Be[471, 0] := 534.701; fTable_Be[471, 1] := 4.28480; fTable_Be[471, 2] := 0.426397;
    fTable_Be[472, 0] := 543.349; fTable_Be[472, 1] := 4.28091; fTable_Be[472, 2] := 0.414215;
    fTable_Be[473, 0] := 552.137; fTable_Be[473, 1] := 4.27707; fTable_Be[473, 2] := 0.402382;
    fTable_Be[474, 0] := 561.068; fTable_Be[474, 1] := 4.27342; fTable_Be[474, 2] := 0.390887;
    fTable_Be[475, 0] := 570.142; fTable_Be[475, 1] := 4.26964; fTable_Be[475, 2] := 0.379297;
    fTable_Be[476, 0] := 579.364; fTable_Be[476, 1] := 4.26575; fTable_Be[476, 2] := 0.368051;
    fTable_Be[477, 0] := 588.735; fTable_Be[477, 1] := 4.26181; fTable_Be[477, 2] := 0.357139;
    fTable_Be[478, 0] := 598.257; fTable_Be[478, 1] := 4.25782; fTable_Be[478, 2] := 0.346550;
    fTable_Be[479, 0] := 607.933; fTable_Be[479, 1] := 4.25382; fTable_Be[479, 2] := 0.336275;
    fTable_Be[480, 0] := 617.766; fTable_Be[480, 1] := 4.24986; fTable_Be[480, 2] := 0.326305;
    fTable_Be[481, 0] := 627.758; fTable_Be[481, 1] := 4.24601; fTable_Be[481, 2] := 0.316630;
    fTable_Be[482, 0] := 637.912; fTable_Be[482, 1] := 4.24229; fTable_Be[482, 2] := 0.307242;
    fTable_Be[483, 0] := 648.229; fTable_Be[483, 1] := 4.23849; fTable_Be[483, 2] := 0.297321;
    fTable_Be[484, 0] := 658.714; fTable_Be[484, 1] := 4.23444; fTable_Be[484, 2] := 0.287720;
    fTable_Be[485, 0] := 669.368; fTable_Be[485, 1] := 4.22972; fTable_Be[485, 2] := 0.278430;
    fTable_Be[486, 0] := 680.195; fTable_Be[486, 1] := 4.22459; fTable_Be[486, 2] := 0.270148;
    fTable_Be[487, 0] := 691.196; fTable_Be[487, 1] := 4.22029; fTable_Be[487, 2] := 0.262802;
    fTable_Be[488, 0] := 702.376; fTable_Be[488, 1] := 4.21661; fTable_Be[488, 2] := 0.255654;
    fTable_Be[489, 0] := 713.736; fTable_Be[489, 1] := 4.21310; fTable_Be[489, 2] := 0.247975;
    fTable_Be[490, 0] := 725.280; fTable_Be[490, 1] := 4.20947; fTable_Be[490, 2] := 0.240525;
    fTable_Be[491, 0] := 737.011; fTable_Be[491, 1] := 4.20574; fTable_Be[491, 2] := 0.233102;
    fTable_Be[492, 0] := 748.932; fTable_Be[492, 1] := 4.20199; fTable_Be[492, 2] := 0.225907;
    fTable_Be[493, 0] := 761.045; fTable_Be[493, 1] := 4.19823; fTable_Be[493, 2] := 0.218934;
    fTable_Be[494, 0] := 773.354; fTable_Be[494, 1] := 4.19446; fTable_Be[494, 2] := 0.212177;
    fTable_Be[495, 0] := 785.863; fTable_Be[495, 1] := 4.19072; fTable_Be[495, 2] := 0.205628;
    fTable_Be[496, 0] := 798.573; fTable_Be[496, 1] := 4.18700; fTable_Be[496, 2] := 0.199281;
    fTable_Be[497, 0] := 811.490; fTable_Be[497, 1] := 4.18331; fTable_Be[497, 2] := 0.193131;
    fTable_Be[498, 0] := 824.615; fTable_Be[498, 1] := 4.17967; fTable_Be[498, 2] := 0.187170;
    fTable_Be[499, 0] := 837.952; fTable_Be[499, 1] := 4.17606; fTable_Be[499, 2] := 0.181392;
    fTable_Be[500, 0] := 851.505; fTable_Be[500, 1] := 4.17249; fTable_Be[500, 2] := 0.175794;
    fTable_Be[501, 0] := 865.278; fTable_Be[501, 1] := 4.16897; fTable_Be[501, 2] := 0.170368;
    fTable_Be[502, 0] := 879.273; fTable_Be[502, 1] := 4.16547; fTable_Be[502, 2] := 0.165110;
    fTable_Be[503, 0] := 893.495; fTable_Be[503, 1] := 4.16203; fTable_Be[503, 2] := 0.160057;
    fTable_Be[504, 0] := 907.946; fTable_Be[504, 1] := 4.15866; fTable_Be[504, 2] := 0.155160;
    fTable_Be[505, 0] := 922.631; fTable_Be[505, 1] := 4.15540; fTable_Be[505, 2] := 0.150411;
    fTable_Be[506, 0] := 937.554; fTable_Be[506, 1] := 4.15220; fTable_Be[506, 2] := 0.145809;
    fTable_Be[507, 0] := 952.719; fTable_Be[507, 1] := 4.14905; fTable_Be[507, 2] := 0.141250;
    fTable_Be[508, 0] := 968.128; fTable_Be[508, 1] := 4.14591; fTable_Be[508, 2] := 0.136834;
    fTable_Be[509, 0] := 983.787; fTable_Be[509, 1] := 4.14280; fTable_Be[509, 2] := 0.132557;
    fTable_Be[510, 0] := 999.699; fTable_Be[510, 1] := 4.13974; fTable_Be[510, 2] := 0.128412;
    fTable_Be[511, 0] := 1015.87; fTable_Be[511, 1] := 4.13672; fTable_Be[511, 2] := 0.124398;
    fTable_Be[512, 0] := 1032.30; fTable_Be[512, 1] := 4.13375; fTable_Be[512, 2] := 0.120509;
    fTable_Be[513, 0] := 1049; fTable_Be[513, 1] := 4.13082; fTable_Be[513, 2] := 0.116741;
    fTable_Be[514, 0] := 1065.96; fTable_Be[514, 1] := 4.12794; fTable_Be[514, 2] := 0.113091;
    fTable_Be[515, 0] := 1083.20; fTable_Be[515, 1] := 4.12511; fTable_Be[515, 2] := 0.109556;
    fTable_Be[516, 0] := 1100.72; fTable_Be[516, 1] := 4.12233; fTable_Be[516, 2] := 0.106131;
    fTable_Be[517, 0] := 1118.53; fTable_Be[517, 1] := 4.11960; fTable_Be[517, 2] := 0.102813;
    fTable_Be[518, 0] := 1136.62; fTable_Be[518, 1] := 4.11692; fTable_Be[518, 2] := 0.0995984;
    fTable_Be[519, 0] := 1155; fTable_Be[519, 1] := 4.11429; fTable_Be[519, 2] := 0.0964847;
    fTable_Be[520, 0] := 1173.68; fTable_Be[520, 1] := 4.11170; fTable_Be[520, 2] := 0.0934681;
    fTable_Be[521, 0] := 1192.67; fTable_Be[521, 1] := 4.10917; fTable_Be[521, 2] := 0.0905461;
    fTable_Be[522, 0] := 1211.96; fTable_Be[522, 1] := 4.10668; fTable_Be[522, 2] := 0.0877153;
    fTable_Be[523, 0] := 1231.56; fTable_Be[523, 1] := 4.10424; fTable_Be[523, 2] := 0.0849730;
    fTable_Be[524, 0] := 1251.48; fTable_Be[524, 1] := 4.10185; fTable_Be[524, 2] := 0.0823165;
    fTable_Be[525, 0] := 1271.72; fTable_Be[525, 1] := 4.09951; fTable_Be[525, 2] := 0.0797430;
    fTable_Be[526, 0] := 1292.29; fTable_Be[526, 1] := 4.09722; fTable_Be[526, 2] := 0.0772499;
    fTable_Be[527, 0] := 1313.19; fTable_Be[527, 1] := 4.09497; fTable_Be[527, 2] := 0.0748349;
    fTable_Be[528, 0] := 1334.43; fTable_Be[528, 1] := 4.09277; fTable_Be[528, 2] := 0.0724952;
    fTable_Be[529, 0] := 1356.01; fTable_Be[529, 1] := 4.09061; fTable_Be[529, 2] := 0.0702288;
    fTable_Be[530, 0] := 1377.95; fTable_Be[530, 1] := 4.08851; fTable_Be[530, 2] := 0.0680301;
    fTable_Be[531, 0] := 1400.23; fTable_Be[531, 1] := 4.08644; fTable_Be[531, 2] := 0.0659001;
    fTable_Be[532, 0] := 1422.88; fTable_Be[532, 1] := 4.08442; fTable_Be[532, 2] := 0.0638369;
    fTable_Be[533, 0] := 1445.90; fTable_Be[533, 1] := 4.08245; fTable_Be[533, 2] := 0.0618382;
    fTable_Be[534, 0] := 1469.28; fTable_Be[534, 1] := 4.08052; fTable_Be[534, 2] := 0.0599022;
    fTable_Be[535, 0] := 1493.05; fTable_Be[535, 1] := 4.07864; fTable_Be[535, 2] := 0.0580268;
    fTable_Be[536, 0] := 1517.20; fTable_Be[536, 1] := 4.07683; fTable_Be[536, 2] := 0.0562100;
    fTable_Be[537, 0] := 1541.73; fTable_Be[537, 1] := 4.07504; fTable_Be[537, 2] := 0.0543948;
    fTable_Be[538, 0] := 1566.67; fTable_Be[538, 1] := 4.07327; fTable_Be[538, 2] := 0.0526382;
    fTable_Be[539, 0] := 1592.01; fTable_Be[539, 1] := 4.07153; fTable_Be[539, 2] := 0.0509382;
    fTable_Be[540, 0] := 1617.76; fTable_Be[540, 1] := 4.06982; fTable_Be[540, 2] := 0.0492933;
    fTable_Be[541, 0] := 1643.93; fTable_Be[541, 1] := 4.06814; fTable_Be[541, 2] := 0.0477014;
    fTable_Be[542, 0] := 1670.52; fTable_Be[542, 1] := 4.06650; fTable_Be[542, 2] := 0.0461609;
    fTable_Be[543, 0] := 1697.53; fTable_Be[543, 1] := 4.06489; fTable_Be[543, 2] := 0.0446702;
    fTable_Be[544, 0] := 1724.99; fTable_Be[544, 1] := 4.06331; fTable_Be[544, 2] := 0.0432276;
    fTable_Be[545, 0] := 1752.89; fTable_Be[545, 1] := 4.06176; fTable_Be[545, 2] := 0.0418316;
    fTable_Be[546, 0] := 1781.24; fTable_Be[546, 1] := 4.06025; fTable_Be[546, 2] := 0.0404807;
    fTable_Be[547, 0] := 1810.05; fTable_Be[547, 1] := 4.05877; fTable_Be[547, 2] := 0.0391734;
    fTable_Be[548, 0] := 1839.33; fTable_Be[548, 1] := 4.05733; fTable_Be[548, 2] := 0.0379083;
    fTable_Be[549, 0] := 1869.08; fTable_Be[549, 1] := 4.05592; fTable_Be[549, 2] := 0.0366841;
    fTable_Be[550, 0] := 1899.31; fTable_Be[550, 1] := 4.05453; fTable_Be[550, 2] := 0.0354994;
    fTable_Be[551, 0] := 1930.03; fTable_Be[551, 1] := 4.05319; fTable_Be[551, 2] := 0.0343530;
    fTable_Be[552, 0] := 1961.25; fTable_Be[552, 1] := 4.05187; fTable_Be[552, 2] := 0.0332436;
    fTable_Be[553, 0] := 1992.97; fTable_Be[553, 1] := 4.05059; fTable_Be[553, 2] := 0.0321700;
    fTable_Be[554, 0] := 2025.20; fTable_Be[554, 1] := 4.04935; fTable_Be[554, 2] := 0.0311311;
    fTable_Be[555, 0] := 2057.96; fTable_Be[555, 1] := 4.04813; fTable_Be[555, 2] := 0.0300957;
    fTable_Be[556, 0] := 2091.24; fTable_Be[556, 1] := 4.04693; fTable_Be[556, 2] := 0.0290947;
    fTable_Be[557, 0] := 2125.07; fTable_Be[557, 1] := 4.04575; fTable_Be[557, 2] := 0.0281270;
    fTable_Be[558, 0] := 2159.44; fTable_Be[558, 1] := 4.04460; fTable_Be[558, 2] := 0.0271914;
    fTable_Be[559, 0] := 2194.37; fTable_Be[559, 1] := 4.04346; fTable_Be[559, 2] := 0.0262870;
    fTable_Be[560, 0] := 2229.86; fTable_Be[560, 1] := 4.04236; fTable_Be[560, 2] := 0.0254127;
    fTable_Be[561, 0] := 2265.93; fTable_Be[561, 1] := 4.04127; fTable_Be[561, 2] := 0.0245675;
    fTable_Be[562, 0] := 2302.57; fTable_Be[562, 1] := 4.04021; fTable_Be[562, 2] := 0.0237503;
    fTable_Be[563, 0] := 2339.82; fTable_Be[563, 1] := 4.03918; fTable_Be[563, 2] := 0.0229604;
    fTable_Be[564, 0] := 2377.66; fTable_Be[564, 1] := 4.03817; fTable_Be[564, 2] := 0.0221967;
    fTable_Be[565, 0] := 2416.12; fTable_Be[565, 1] := 4.03718; fTable_Be[565, 2] := 0.0214584;
    fTable_Be[566, 0] := 2455.20; fTable_Be[566, 1] := 4.03621; fTable_Be[566, 2] := 0.0207447;
    fTable_Be[567, 0] := 2494.91; fTable_Be[567, 1] := 4.03527; fTable_Be[567, 2] := 0.0200547;
    fTable_Be[568, 0] := 2535.26; fTable_Be[568, 1] := 4.03435; fTable_Be[568, 2] := 0.0193877;
    fTable_Be[569, 0] := 2576.27; fTable_Be[569, 1] := 4.03345; fTable_Be[569, 2] := 0.0187429;
    fTable_Be[570, 0] := 2617.94; fTable_Be[570, 1] := 4.03257; fTable_Be[570, 2] := 0.0181195;
    fTable_Be[571, 0] := 2660.28; fTable_Be[571, 1] := 4.03171; fTable_Be[571, 2] := 0.0175168;
    fTable_Be[572, 0] := 2703.31; fTable_Be[572, 1] := 4.03088; fTable_Be[572, 2] := 0.0169342;
    fTable_Be[573, 0] := 2747.03; fTable_Be[573, 1] := 4.03006; fTable_Be[573, 2] := 0.0163709;
    fTable_Be[574, 0] := 2791.46; fTable_Be[574, 1] := 4.02926; fTable_Be[574, 2] := 0.0158264;
    fTable_Be[575, 0] := 2836.61; fTable_Be[575, 1] := 4.02849; fTable_Be[575, 2] := 0.0153000;
    fTable_Be[576, 0] := 2882.49; fTable_Be[576, 1] := 4.02773; fTable_Be[576, 2] := 0.0147911;
    fTable_Be[577, 0] := 2929.11; fTable_Be[577, 1] := 4.02700; fTable_Be[577, 2] := 0.0142992;
    fTable_Be[578, 0] := 2976.49; fTable_Be[578, 1] := 4.02628; fTable_Be[578, 2] := 0.0138236;
    fTable_Be[579, 0] := 3024.63; fTable_Be[579, 1] := 4.02559; fTable_Be[579, 2] := 0.0133638;
    fTable_Be[580, 0] := 3073.55; fTable_Be[580, 1] := 4.02491; fTable_Be[580, 2] := 0.0129072;
    fTable_Be[581, 0] := 3123.26; fTable_Be[581, 1] := 4.02424; fTable_Be[581, 2] := 0.0124663;
    fTable_Be[582, 0] := 3173.78; fTable_Be[582, 1] := 4.02359; fTable_Be[582, 2] := 0.0120403;
    fTable_Be[583, 0] := 3225.11; fTable_Be[583, 1] := 4.02295; fTable_Be[583, 2] := 0.0116290;
    fTable_Be[584, 0] := 3277.28; fTable_Be[584, 1] := 4.02233; fTable_Be[584, 2] := 0.0112317;
    fTable_Be[585, 0] := 3330.29; fTable_Be[585, 1] := 4.02172; fTable_Be[585, 2] := 0.0108480;
    fTable_Be[586, 0] := 3384.15; fTable_Be[586, 1] := 4.02113; fTable_Be[586, 2] := 0.0104774;
    fTable_Be[587, 0] := 3438.89; fTable_Be[587, 1] := 4.02055; fTable_Be[587, 2] := 0.0101194;
    fTable_Be[588, 0] := 3494.51; fTable_Be[588, 1] := 4.01998; fTable_Be[588, 2] := 0.00977365;
    fTable_Be[589, 0] := 3551.03; fTable_Be[589, 1] := 4.01943; fTable_Be[589, 2] := 0.00943974;
    fTable_Be[590, 0] := 3608.46; fTable_Be[590, 1] := 4.01890; fTable_Be[590, 2] := 0.00911724;
    fTable_Be[591, 0] := 3666.83; fTable_Be[591, 1] := 4.01837; fTable_Be[591, 2] := 0.00880575;
    fTable_Be[592, 0] := 3726.13; fTable_Be[592, 1] := 4.01786; fTable_Be[592, 2] := 0.00850491;
    fTable_Be[593, 0] := 3786.40; fTable_Be[593, 1] := 4.01736; fTable_Be[593, 2] := 0.00821432;
    fTable_Be[594, 0] := 3847.64; fTable_Be[594, 1] := 4.01688; fTable_Be[594, 2] := 0.00793369;
    fTable_Be[595, 0] := 3909.88; fTable_Be[595, 1] := 4.01641; fTable_Be[595, 2] := 0.00766264;
    fTable_Be[596, 0] := 3973.12; fTable_Be[596, 1] := 4.01595; fTable_Be[596, 2] := 0.00740085;
    fTable_Be[597, 0] := 4037.38; fTable_Be[597, 1] := 4.01550; fTable_Be[597, 2] := 0.00714801;
    fTable_Be[598, 0] := 4102.68; fTable_Be[598, 1] := 4.01506; fTable_Be[598, 2] := 0.00690380;
    fTable_Be[599, 0] := 4169.04; fTable_Be[599, 1] := 4.01464; fTable_Be[599, 2] := 0.00666401;
    fTable_Be[600, 0] := 4236.47; fTable_Be[600, 1] := 4.01423; fTable_Be[600, 2] := 0.00643256;
    fTable_Be[601, 0] := 4304.99; fTable_Be[601, 1] := 4.01382; fTable_Be[601, 2] := 0.00620915;
    fTable_Be[602, 0] := 4374.62; fTable_Be[602, 1] := 4.01343; fTable_Be[602, 2] := 0.00599350;
    fTable_Be[603, 0] := 4445.37; fTable_Be[603, 1] := 4.01304; fTable_Be[603, 2] := 0.00578535;
    fTable_Be[604, 0] := 4517.27; fTable_Be[604, 1] := 4.01267; fTable_Be[604, 2] := 0.00558442;
    fTable_Be[605, 0] := 4590.34; fTable_Be[605, 1] := 4.01230; fTable_Be[605, 2] := 0.00539045;
    fTable_Be[606, 0] := 4664.58; fTable_Be[606, 1] := 4.01195; fTable_Be[606, 2] := 0.00520323;
    fTable_Be[607, 0] := 4740.03; fTable_Be[607, 1] := 4.01160; fTable_Be[607, 2] := 0.00502252;
    fTable_Be[608, 0] := 4816.70; fTable_Be[608, 1] := 4.01126; fTable_Be[608, 2] := 0.00484809;
    fTable_Be[609, 0] := 4894.60; fTable_Be[609, 1] := 4.01093; fTable_Be[609, 2] := 0.00467971;
    fTable_Be[610, 0] := 4973.77; fTable_Be[610, 1] := 4.01061; fTable_Be[610, 2] := 0.00451716;
    fTable_Be[611, 0] := 5054.21; fTable_Be[611, 1] := 4.01030; fTable_Be[611, 2] := 0.00436028;
    fTable_Be[612, 0] := 5135.96; fTable_Be[612, 1] := 4.01000; fTable_Be[612, 2] := 0.00420884;
    fTable_Be[613, 0] := 5219.03; fTable_Be[613, 1] := 4.00970; fTable_Be[613, 2] := 0.00406267;
    fTable_Be[614, 0] := 5303.45; fTable_Be[614, 1] := 4.00941; fTable_Be[614, 2] := 0.00391977;
    fTable_Be[615, 0] := 5389.23; fTable_Be[615, 1] := 4.00913; fTable_Be[615, 2] := 0.00378191;
    fTable_Be[616, 0] := 5476.39; fTable_Be[616, 1] := 4.00886; fTable_Be[616, 2] := 0.00364888;
    fTable_Be[617, 0] := 5564.97; fTable_Be[617, 1] := 4.00860; fTable_Be[617, 2] := 0.00352054;
    fTable_Be[618, 0] := 5654.98; fTable_Be[618, 1] := 4.00834; fTable_Be[618, 2] := 0.00339671;
    fTable_Be[619, 0] := 5746.44; fTable_Be[619, 1] := 4.00808; fTable_Be[619, 2] := 0.00327724;
    fTable_Be[620, 0] := 5839.39; fTable_Be[620, 1] := 4.00784; fTable_Be[620, 2] := 0.00316197;
    fTable_Be[621, 0] := 5933.83; fTable_Be[621, 1] := 4.00760; fTable_Be[621, 2] := 0.00305075;
    fTable_Be[622, 0] := 6029.81; fTable_Be[622, 1] := 4.00737; fTable_Be[622, 2] := 0.00294344;
    fTable_Be[623, 0] := 6127.33; fTable_Be[623, 1] := 4.00714; fTable_Be[623, 2] := 0.00283992;
    fTable_Be[624, 0] := 6226.44; fTable_Be[624, 1] := 4.00692; fTable_Be[624, 2] := 0.00274003;
    fTable_Be[625, 0] := 6327.15; fTable_Be[625, 1] := 4.00671; fTable_Be[625, 2] := 0.00264365;
    fTable_Be[626, 0] := 6429.48; fTable_Be[626, 1] := 4.00650; fTable_Be[626, 2] := 0.00254975;
    fTable_Be[627, 0] := 6533.48; fTable_Be[627, 1] := 4.00630; fTable_Be[627, 2] := 0.00245918;
    fTable_Be[628, 0] := 6639.15; fTable_Be[628, 1] := 4.00610; fTable_Be[628, 2] := 0.00237183;
    fTable_Be[629, 0] := 6746.53; fTable_Be[629, 1] := 4.00591; fTable_Be[629, 2] := 0.00228759;
    fTable_Be[630, 0] := 6855.65; fTable_Be[630, 1] := 4.00572; fTable_Be[630, 2] := 0.00220633;
    fTable_Be[631, 0] := 6966.54; fTable_Be[631, 1] := 4.00554; fTable_Be[631, 2] := 0.00212796;
    fTable_Be[632, 0] := 7079.21; fTable_Be[632, 1] := 4.00536; fTable_Be[632, 2] := 0.00205238;
    fTable_Be[633, 0] := 7193.71; fTable_Be[633, 1] := 4.00519; fTable_Be[633, 2] := 0.00197947;
    fTable_Be[634, 0] := 7310.07; fTable_Be[634, 1] := 4.00502; fTable_Be[634, 2] := 0.00190916;
    fTable_Be[635, 0] := 7428.30; fTable_Be[635, 1] := 4.00485; fTable_Be[635, 2] := 0.00184135;
    fTable_Be[636, 0] := 7548.45; fTable_Be[636, 1] := 4.00469; fTable_Be[636, 2] := 0.00177595;
    fTable_Be[637, 0] := 7670.54; fTable_Be[637, 1] := 4.00454; fTable_Be[637, 2] := 0.00171287;
    fTable_Be[638, 0] := 7794.60; fTable_Be[638, 1] := 4.00439; fTable_Be[638, 2] := 0.00165202;
    fTable_Be[639, 0] := 7920.68; fTable_Be[639, 1] := 4.00424; fTable_Be[639, 2] := 0.00159334;
    fTable_Be[640, 0] := 8048.79; fTable_Be[640, 1] := 4.00410; fTable_Be[640, 2] := 0.00153675;
    fTable_Be[641, 0] := 8178.97; fTable_Be[641, 1] := 4.00396; fTable_Be[641, 2] := 0.00148216;
    fTable_Be[642, 0] := 8311.26; fTable_Be[642, 1] := 4.00383; fTable_Be[642, 2] := 0.00142952;
    fTable_Be[643, 0] := 8445.68; fTable_Be[643, 1] := 4.00370; fTable_Be[643, 2] := 0.00137819;
    fTable_Be[644, 0] := 8582.29; fTable_Be[644, 1] := 4.00357; fTable_Be[644, 2] := 0.00132870;
    fTable_Be[645, 0] := 8721.10; fTable_Be[645, 1] := 4.00345; fTable_Be[645, 2] := 0.00128099;
    fTable_Be[646, 0] := 8862.16; fTable_Be[646, 1] := 4.00333; fTable_Be[646, 2] := 0.00123499;
    fTable_Be[647, 0] := 9005.49; fTable_Be[647, 1] := 4.00321; fTable_Be[647, 2] := 0.00119064;
    fTable_Be[648, 0] := 9151.15; fTable_Be[648, 1] := 4.00310; fTable_Be[648, 2] := 0.00114789;
    fTable_Be[649, 0] := 9299.16; fTable_Be[649, 1] := 4.00299; fTable_Be[649, 2] := 0.00110667;
    fTable_Be[650, 0] := 9449.57; fTable_Be[650, 1] := 4.00288; fTable_Be[650, 2] := 0.00106693;
    fTable_Be[651, 0] := 9602.41; fTable_Be[651, 1] := 4.00277; fTable_Be[651, 2] := 0.00102862;
    fTable_Be[652, 0] := 9757.72; fTable_Be[652, 1] := 4.00267; fTable_Be[652, 2] := 0.000991686;
    fTable_Be[653, 0] := 9915.54; fTable_Be[653, 1] := 4.00257; fTable_Be[653, 2] := 0.000956077;
    fTable_Be[654, 0] := 10075.9; fTable_Be[654, 1] := 4.00248; fTable_Be[654, 2] := 0.000921746;
    fTable_Be[655, 0] := 10238.9; fTable_Be[655, 1] := 4.00238; fTable_Be[655, 2] := 0.000888646;
    fTable_Be[656, 0] := 10404.5; fTable_Be[656, 1] := 4.00229; fTable_Be[656, 2] := 0.000856737;
    fTable_Be[657, 0] := 10572.8; fTable_Be[657, 1] := 4.00221; fTable_Be[657, 2] := 0.000825973;
    fTable_Be[658, 0] := 10743.8; fTable_Be[658, 1] := 4.00212; fTable_Be[658, 2] := 0.000796314;
    fTable_Be[659, 0] := 10917.6; fTable_Be[659, 1] := 4.00204; fTable_Be[659, 2] := 0.000767721;
    fTable_Be[660, 0] := 11094.1; fTable_Be[660, 1] := 4.00196; fTable_Be[660, 2] := 0.000740154;
    fTable_Be[661, 0] := 11273.6; fTable_Be[661, 1] := 4.00188; fTable_Be[661, 2] := 0.000713574;
    fTable_Be[662, 0] := 11455.9; fTable_Be[662, 1] := 4.00180; fTable_Be[662, 2] := 0.000687952;
    fTable_Be[663, 0] := 11641.2; fTable_Be[663, 1] := 4.00173; fTable_Be[663, 2] := 0.000663249;
    fTable_Be[664, 0] := 11829.5; fTable_Be[664, 1] := 4.00165; fTable_Be[664, 2] := 0.000639433;
    fTable_Be[665, 0] := 12020.8; fTable_Be[665, 1] := 4.00158; fTable_Be[665, 2] := 0.000616473;
    fTable_Be[666, 0] := 12215.3; fTable_Be[666, 1] := 4.00152; fTable_Be[666, 2] := 0.000594337;
    fTable_Be[667, 0] := 12412.8; fTable_Be[667, 1] := 4.00145; fTable_Be[667, 2] := 0.000572994;
    fTable_Be[668, 0] := 12613.6; fTable_Be[668, 1] := 4.00139; fTable_Be[668, 2] := 0.000552174;
    fTable_Be[669, 0] := 12817.6; fTable_Be[669, 1] := 4.00132; fTable_Be[669, 2] := 0.000532111;
    fTable_Be[670, 0] := 13024.9; fTable_Be[670, 1] := 4.00126; fTable_Be[670, 2] := 0.000512776;
    fTable_Be[671, 0] := 13235.6; fTable_Be[671, 1] := 4.00120; fTable_Be[671, 2] := 0.000494145;
    fTable_Be[672, 0] := 13449.7; fTable_Be[672, 1] := 4.00115; fTable_Be[672, 2] := 0.000476188;
    fTable_Be[673, 0] := 13667.2; fTable_Be[673, 1] := 4.00109; fTable_Be[673, 2] := 0.000458886;
    fTable_Be[674, 0] := 13888.3; fTable_Be[674, 1] := 4.00104; fTable_Be[674, 2] := 0.000442212;
    fTable_Be[675, 0] := 14112.9; fTable_Be[675, 1] := 4.00098; fTable_Be[675, 2] := 0.000426144;
    fTable_Be[676, 0] := 14341.2; fTable_Be[676, 1] := 4.00093; fTable_Be[676, 2] := 0.000410660;
    fTable_Be[677, 0] := 14573.1; fTable_Be[677, 1] := 4.00088; fTable_Be[677, 2] := 0.000395739;
    fTable_Be[678, 0] := 14808.8; fTable_Be[678, 1] := 4.00083; fTable_Be[678, 2] := 0.000381358;
    fTable_Be[679, 0] := 15048.3; fTable_Be[679, 1] := 4.00079; fTable_Be[679, 2] := 0.000367502;
    fTable_Be[680, 0] := 15291.7; fTable_Be[680, 1] := 4.00074; fTable_Be[680, 2] := 0.000354148;
    fTable_Be[681, 0] := 15539.1; fTable_Be[681, 1] := 4.00070; fTable_Be[681, 2] := 0.000341280;
    fTable_Be[682, 0] := 15790.4; fTable_Be[682, 1] := 4.00065; fTable_Be[682, 2] := 0.000328880;
    fTable_Be[683, 0] := 16045.8; fTable_Be[683, 1] := 4.00061; fTable_Be[683, 2] := 0.000316929;
    fTable_Be[684, 0] := 16305.3; fTable_Be[684, 1] := 4.00057; fTable_Be[684, 2] := 0.000305413;
    fTable_Be[685, 0] := 16569.1; fTable_Be[685, 1] := 4.00053; fTable_Be[685, 2] := 0.000294207;
    fTable_Be[686, 0] := 16837.0; fTable_Be[686, 1] := 4.00049; fTable_Be[686, 2] := 0.000283413;
    fTable_Be[687, 0] := 17109.4; fTable_Be[687, 1] := 4.00046; fTable_Be[687, 2] := 0.000273015;
    fTable_Be[688, 0] := 17386.1; fTable_Be[688, 1] := 4.00042; fTable_Be[688, 2] := 0.000262998;
    fTable_Be[689, 0] := 17667.3; fTable_Be[689, 1] := 4.00039; fTable_Be[689, 2] := 0.000253348;
    fTable_Be[690, 0] := 17953.1; fTable_Be[690, 1] := 4.00035; fTable_Be[690, 2] := 0.000244052;
    fTable_Be[691, 0] := 18243.4; fTable_Be[691, 1] := 4.00032; fTable_Be[691, 2] := 0.000235098;
    fTable_Be[692, 0] := 18538.5; fTable_Be[692, 1] := 4.00029; fTable_Be[692, 2] := 0.000226472;
    fTable_Be[693, 0] := 18838.4; fTable_Be[693, 1] := 4.00026; fTable_Be[693, 2] := 0.000218163;
    fTable_Be[694, 0] := 19143.0; fTable_Be[694, 1] := 4.00023; fTable_Be[694, 2] := 0.000210159;
    fTable_Be[695, 0] := 19452.7; fTable_Be[695, 1] := 4.00020; fTable_Be[695, 2] := 0.000202447;
    fTable_Be[696, 0] := 19767.3; fTable_Be[696, 1] := 4.00017; fTable_Be[696, 2] := 0.000195019;
    fTable_Be[697, 0] := 20087.0; fTable_Be[697, 1] := 4.00014; fTable_Be[697, 2] := 0.000187864;
    fTable_Be[698, 0] := 20411.9; fTable_Be[698, 1] := 4.00011; fTable_Be[698, 2] := 0.000180971;
    fTable_Be[699, 0] := 20742.1; fTable_Be[699, 1] := 4.00009; fTable_Be[699, 2] := 0.000174332;
    fTable_Be[700, 0] := 21077.5; fTable_Be[700, 1] := 4.00006; fTable_Be[700, 2] := 0.000167935;
    fTable_Be[701, 0] := 21418.5; fTable_Be[701, 1] := 4.00004; fTable_Be[701, 2] := 0.000161773;
    fTable_Be[702, 0] := 21764.9; fTable_Be[702, 1] := 4.00001; fTable_Be[702, 2] := 0.000155838;
    fTable_Be[703, 0] := 22116.9; fTable_Be[703, 1] := 3.99999; fTable_Be[703, 2] := 0.000150120;
    fTable_Be[704, 0] := 22474.6; fTable_Be[704, 1] := 3.99997; fTable_Be[704, 2] := 0.000144612;
    fTable_Be[705, 0] := 22838.1; fTable_Be[705, 1] := 3.99995; fTable_Be[705, 2] := 0.000139307;
    fTable_Be[706, 0] := 23207.5; fTable_Be[706, 1] := 3.99992; fTable_Be[706, 2] := 0.000134195;
    fTable_Be[707, 0] := 23582.9; fTable_Be[707, 1] := 3.99990; fTable_Be[707, 2] := 0.000129271;
    fTable_Be[708, 0] := 23964.3; fTable_Be[708, 1] := 3.99988; fTable_Be[708, 2] := 0.000124528;
    fTable_Be[709, 0] := 24351.9; fTable_Be[709, 1] := 3.99986; fTable_Be[709, 2] := 0.000119959;
    fTable_Be[710, 0] := 24745.8; fTable_Be[710, 1] := 3.99985; fTable_Be[710, 2] := 0.000115558;
    fTable_Be[711, 0] := 25146.1; fTable_Be[711, 1] := 3.99983; fTable_Be[711, 2] := 0.000111318;
    fTable_Be[712, 0] := 25552.8; fTable_Be[712, 1] := 3.99981; fTable_Be[712, 2] := 0.000107234;
    fTable_Be[713, 0] := 25966.1; fTable_Be[713, 1] := 3.99979; fTable_Be[713, 2] := 0.000103299;
    fTable_Be[714, 0] := 26386.0; fTable_Be[714, 1] := 3.99978; fTable_Be[714, 2] := 0.0000995092;
    fTable_Be[715, 0] := 26812.8; fTable_Be[715, 1] := 3.99976; fTable_Be[715, 2] := 0.0000958583;
    fTable_Be[716, 0] := 27246.5; fTable_Be[716, 1] := 3.99974; fTable_Be[716, 2] := 0.0000923412;
    fTable_Be[717, 0] := 27687.2; fTable_Be[717, 1] := 3.99973; fTable_Be[717, 2] := 0.0000889532;
    fTable_Be[718, 0] := 28135.0; fTable_Be[718, 1] := 3.99971; fTable_Be[718, 2] := 0.0000856893;
    fTable_Be[719, 0] := 28590.1; fTable_Be[719, 1] := 3.99970; fTable_Be[719, 2] := 0.0000825453;
    fTable_Be[720, 0] := 29052.5; fTable_Be[720, 1] := 3.99969; fTable_Be[720, 2] := 0.0000795168;
    fTable_Be[721, 0] := 29522.4; fTable_Be[721, 1] := 3.99967; fTable_Be[721, 2] := 0.0000765993;
    fTable_Be[722, 0] := 29999.9; fTable_Be[722, 1] := 3.99966; fTable_Be[722, 2] := 0.0000737888;
    fTable_Be[723, 0] := 30000.0; fTable_Be[723, 1] := 3.99966; fTable_Be[723, 2] := 0.0000737882;

